// TIA Portal V20 export
FUNCTION "CollectAlarms" : Void   // FC62, LAD
TITLE = Alarm Collector Unit
// Collects alarms from the respective level and categorises the alarms into the different alarm classes.
// stored: Namespace Unit1, SetENOAutomatically false
   VAR_INPUT
      resetAlarms : Bool;
      disableAlarms : Bool;
   END_VAR
   VAR_OUTPUT
      commandsToUnit : "LUC_typeStateCommands";   // Feedback to the unit
   END_VAR
   VAR CONSTANT
      DelayTime : Time := T#300ms;
      TRUE : Bool := TRUE;
      FALSE : Bool;
   END_VAR
BEGIN

REGION Network 1: Reset Alarms
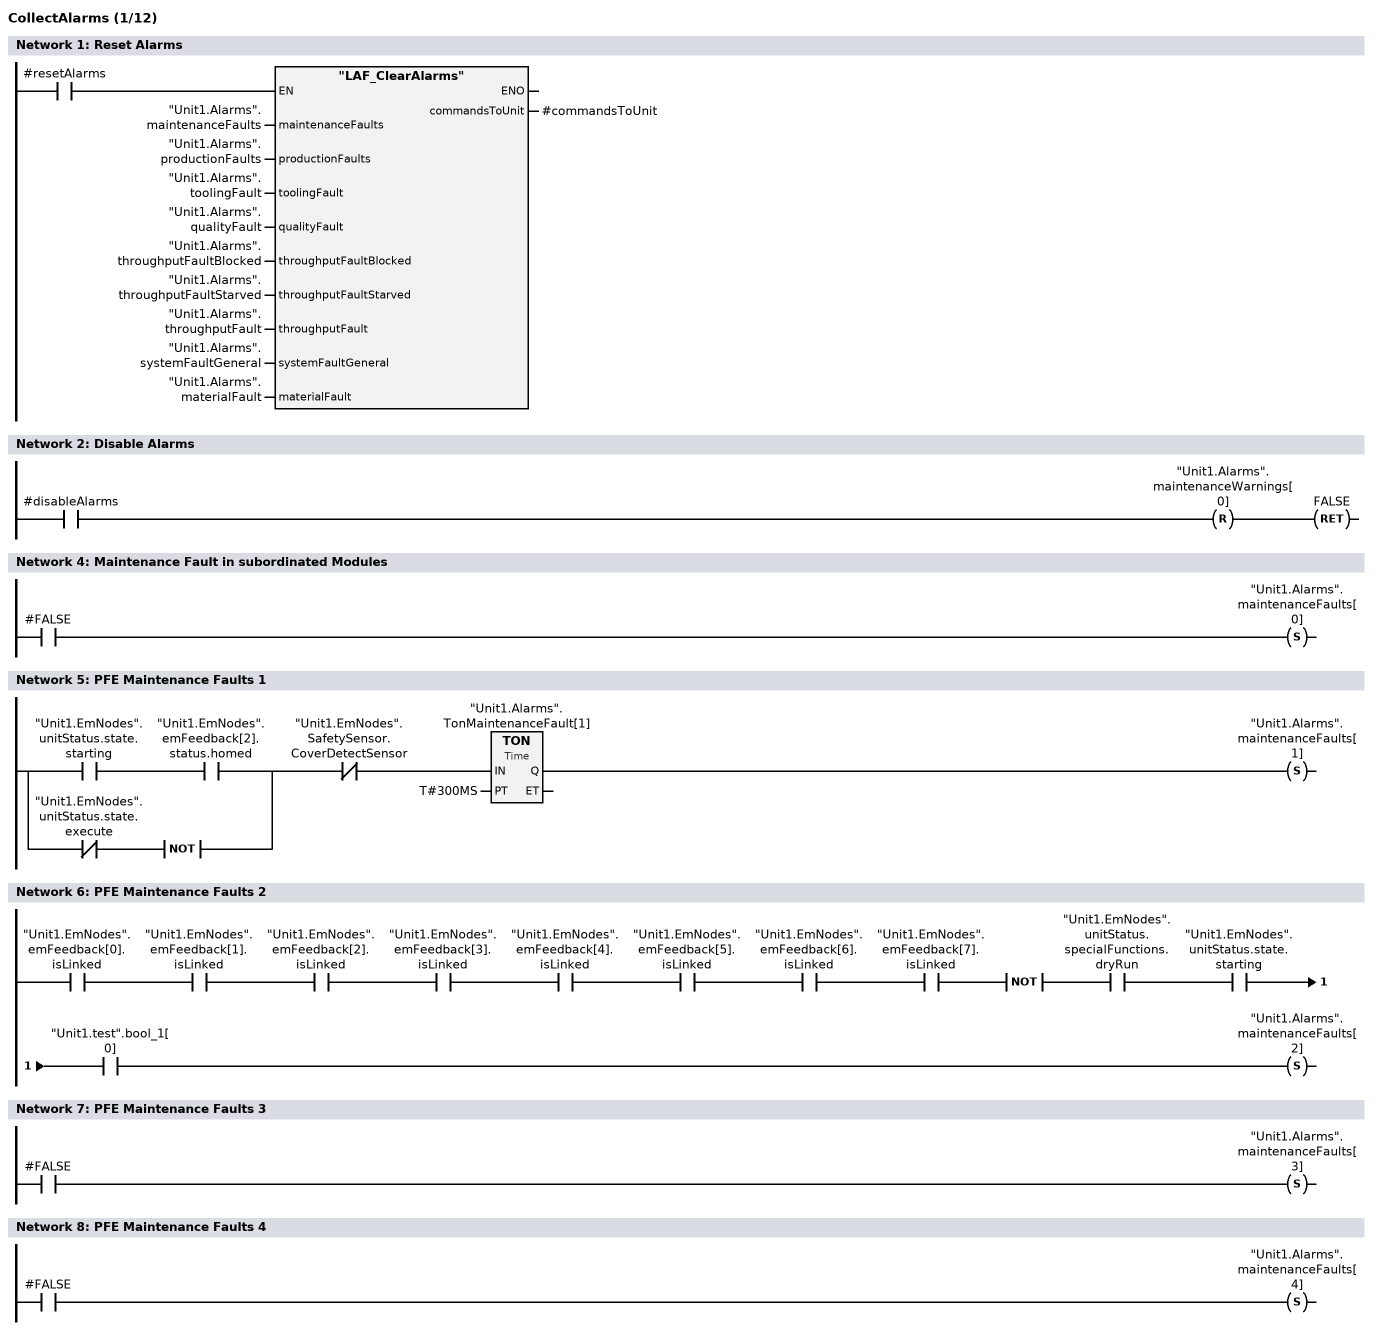
   RUNG wire#powerrail
      Contact( #resetAlarms )
      "LAF_ClearAlarms"(maintenanceFaults := "Unit1.Alarms".maintenanceFaults, productionFaults := "Unit1.Alarms".productionFaults, toolingFault := "Unit1.Alarms".toolingFault, qualityFault := "Unit1.Alarms".qualityFault, throughputFaultBlocked := "Unit1.Alarms".throughputFaultBlocked, throughputFaultStarved := "Unit1.Alarms".throughputFaultStarved, throughputFault := "Unit1.Alarms".throughputFault, systemFaultGeneral := "Unit1.Alarms".systemFaultGeneral, materialFault := "Unit1.Alarms".materialFault, commandsToUnit => #commandsToUnit)
   END_RUNG
   // the same network as SCL:
   IF #resetAlarms THEN
       "LAF_ClearAlarms"(maintenanceFaults := "Unit1.Alarms".maintenanceFaults,
                         productionFaults := "Unit1.Alarms".productionFaults,
                         toolingFault := "Unit1.Alarms".toolingFault,
                         qualityFault := "Unit1.Alarms".qualityFault,
                         throughputFaultBlocked := "Unit1.Alarms".throughputFaultBlocked,
                         throughputFaultStarved := "Unit1.Alarms".throughputFaultStarved,
                         throughputFault := "Unit1.Alarms".throughputFault,
                         systemFaultGeneral := "Unit1.Alarms".systemFaultGeneral,
                         materialFault := "Unit1.Alarms".materialFault,
                         commandsToUnit => #commandsToUnit);
   END_IF;
END_REGION

REGION Network 2: Disable Alarms
   RUNG wire#powerrail
      Contact( #disableAlarms )
      R_Coil( "Unit1.Alarms".maintenanceWarnings[0] )
      ReturnCoil( FALSE )
   END_RUNG
   // the same network as SCL:
   IF #disableAlarms THEN
       "Unit1.Alarms".maintenanceWarnings[0] := FALSE;
       ENO := FALSE;
       RETURN;
   END_IF;
END_REGION

REGION Network 3: *************** Fault ************************
END_REGION

REGION Network 4: Maintenance Fault in subordinated Modules
   RUNG wire#powerrail
      Contact( #FALSE )
      S_Coil( "Unit1.Alarms".maintenanceFaults[0] )
   END_RUNG
   // the same network as SCL:
   IF #FALSE THEN "Unit1.Alarms".maintenanceFaults[0] := TRUE; END_IF;
END_REGION

REGION Network 5: PFE Maintenance Faults 1
   RUNG wire#powerrail
      Contact( "Unit1.EmNodes".unitStatus.state.starting )
      Contact( "Unit1.EmNodes".emFeedback[2].status.homed )
      wire#w1
      I_Contact( "Unit1.EmNodes".SafetySensor.CoverDetectSensor )
      { S7_Templates := "time_type := Time" } "Unit1.Alarms".TonMaintenanceFault[1].TON(pt := T#300MS, et =>)
      S_Coil( "Unit1.Alarms".maintenanceFaults[1] )
   END_RUNG
   RUNG wire#powerrail
      I_Contact( "Unit1.EmNodes".unitStatus.state.execute )
      Not()
   END_RUNG wire#w1
   // the same network as SCL:
   "Unit1.Alarms".TonMaintenanceFault[1].TON(IN := (("Unit1.EmNodes".unitStatus.state.starting AND "Unit1.EmNodes".emFeedback[2].status.homed) OR NOT (NOT "Unit1.EmNodes".unitStatus.state.execute)) AND NOT "Unit1.EmNodes".SafetySensor.CoverDetectSensor,
                           PT := T#300MS);
   IF "Unit1.Alarms".TonMaintenanceFault[1].Q THEN "Unit1.Alarms".maintenanceFaults[1] := TRUE; END_IF;
END_REGION

REGION Network 6: PFE Maintenance Faults 2
   RUNG wire#powerrail
      Contact( "Unit1.EmNodes".emFeedback[0].isLinked )
      Contact( "Unit1.EmNodes".emFeedback[1].isLinked )
      Contact( "Unit1.EmNodes".emFeedback[2].isLinked )
      Contact( "Unit1.EmNodes".emFeedback[3].isLinked )
      Contact( "Unit1.EmNodes".emFeedback[4].isLinked )
      Contact( "Unit1.EmNodes".emFeedback[5].isLinked )
      Contact( "Unit1.EmNodes".emFeedback[6].isLinked )
      Contact( "Unit1.EmNodes".emFeedback[7].isLinked )
      Not()
      Contact( "Unit1.EmNodes".unitStatus.specialFunctions.dryRun )
      Contact( "Unit1.EmNodes".unitStatus.state.starting )
      Contact( "Unit1.test".bool_1[0] )
      S_Coil( "Unit1.Alarms".maintenanceFaults[2] )
   END_RUNG
   // the same network as SCL:
   IF NOT ("Unit1.EmNodes".emFeedback[0].isLinked AND "Unit1.EmNodes".emFeedback[1].isLinked AND "Unit1.EmNodes".emFeedback[2].isLinked AND "Unit1.EmNodes".emFeedback[3].isLinked AND "Unit1.EmNodes".emFeedback[4].isLinked AND "Unit1.EmNodes".emFeedback[5].isLinked AND "Unit1.EmNodes".emFeedback[6].isLinked AND "Unit1.EmNodes".emFeedback[7].isLinked) AND "Unit1.EmNodes".unitStatus.specialFunctions.dryRun AND "Unit1.EmNodes".unitStatus.state.starting AND "Unit1.test".bool_1[0] THEN
       "Unit1.Alarms".maintenanceFaults[2] := TRUE;
   END_IF;
END_REGION

REGION Network 7: PFE Maintenance Faults 3
   RUNG wire#powerrail
      Contact( #FALSE )
      S_Coil( "Unit1.Alarms".maintenanceFaults[3] )
   END_RUNG
   // the same network as SCL:
   IF #FALSE THEN "Unit1.Alarms".maintenanceFaults[3] := TRUE; END_IF;
END_REGION

REGION Network 8: PFE Maintenance Faults 4
   RUNG wire#powerrail
      Contact( #FALSE )
      S_Coil( "Unit1.Alarms".maintenanceFaults[4] )
   END_RUNG
   // the same network as SCL:
   IF #FALSE THEN "Unit1.Alarms".maintenanceFaults[4] := TRUE; END_IF;
END_REGION

REGION Network 9: PFE Maintenance Faults 5
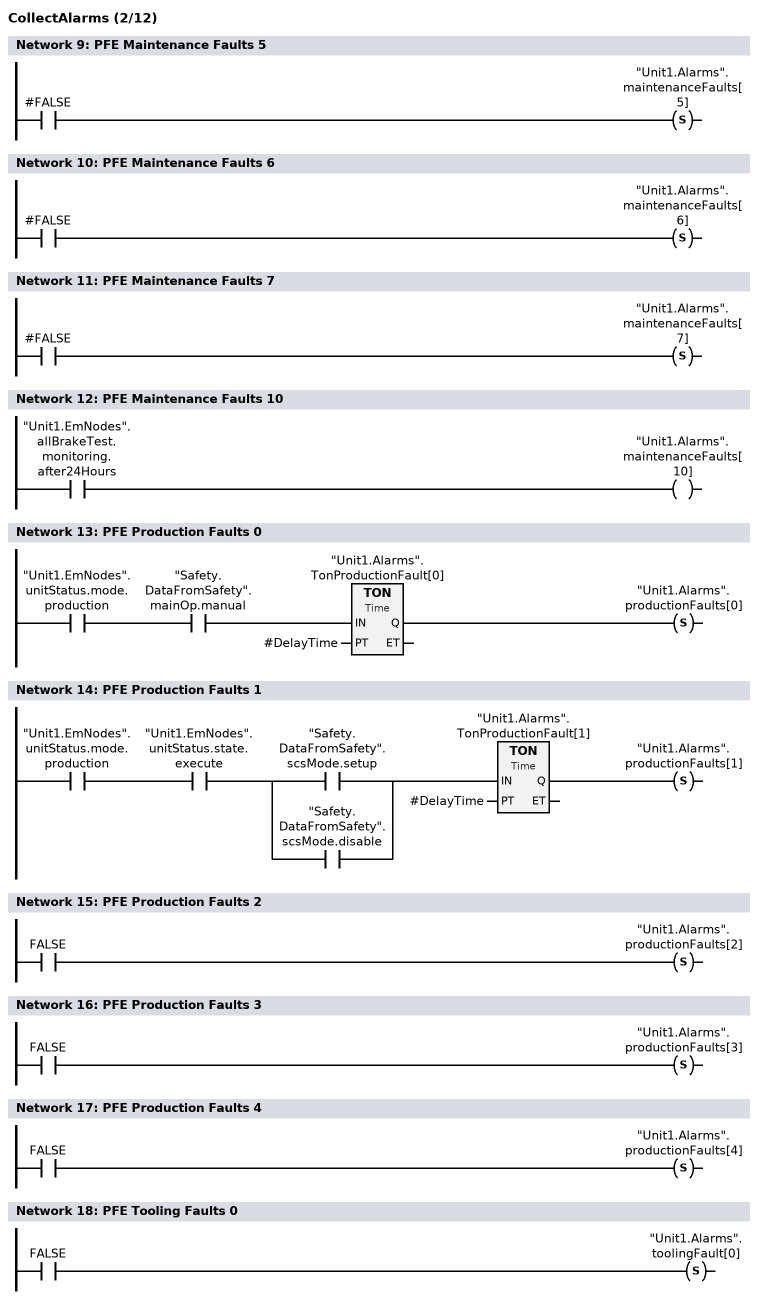
   RUNG wire#powerrail
      Contact( #FALSE )
      S_Coil( "Unit1.Alarms".maintenanceFaults[5] )
   END_RUNG
   // the same network as SCL:
   IF #FALSE THEN "Unit1.Alarms".maintenanceFaults[5] := TRUE; END_IF;
END_REGION

REGION Network 10: PFE Maintenance Faults 6
   RUNG wire#powerrail
      Contact( #FALSE )
      S_Coil( "Unit1.Alarms".maintenanceFaults[6] )
   END_RUNG
   // the same network as SCL:
   IF #FALSE THEN "Unit1.Alarms".maintenanceFaults[6] := TRUE; END_IF;
END_REGION

REGION Network 11: PFE Maintenance Faults 7
   RUNG wire#powerrail
      Contact( #FALSE )
      S_Coil( "Unit1.Alarms".maintenanceFaults[7] )
   END_RUNG
   // the same network as SCL:
   IF #FALSE THEN "Unit1.Alarms".maintenanceFaults[7] := TRUE; END_IF;
END_REGION

REGION Network 12: PFE Maintenance Faults 10
   RUNG wire#powerrail
      Contact( "Unit1.EmNodes".allBrakeTest.monitoring.after24Hours )
      Coil( "Unit1.Alarms".maintenanceFaults[10] )
   END_RUNG
   // the same network as SCL:
   "Unit1.Alarms".maintenanceFaults[10] := "Unit1.EmNodes".allBrakeTest.monitoring.after24Hours;
END_REGION

REGION Network 13: PFE Production Faults 0
   RUNG wire#powerrail
      Contact( "Unit1.EmNodes".unitStatus.mode.production )
      Contact( "Safety.DataFromSafety".mainOp.manual )
      { S7_Templates := "time_type := Time" } "Unit1.Alarms".TonProductionFault[0].TON(pt := #DelayTime, et =>)
      S_Coil( "Unit1.Alarms".productionFaults[0] )
   END_RUNG
   // the same network as SCL:
   "Unit1.Alarms".TonProductionFault[0].TON(IN := "Unit1.EmNodes".unitStatus.mode.production AND "Safety.DataFromSafety".mainOp.manual,
                           PT := #DelayTime);
   IF "Unit1.Alarms".TonProductionFault[0].Q THEN "Unit1.Alarms".productionFaults[0] := TRUE; END_IF;
END_REGION

REGION Network 14: PFE Production Faults 1
   RUNG wire#powerrail
      Contact( "Unit1.EmNodes".unitStatus.mode.production )
      Contact( "Unit1.EmNodes".unitStatus.state.execute )
      wire#w1
      Contact( "Safety.DataFromSafety".scsMode.setup )
      wire#w2
      { S7_Templates := "time_type := Time" } "Unit1.Alarms".TonProductionFault[1].TON(pt := #DelayTime, et =>)
      S_Coil( "Unit1.Alarms".productionFaults[1] )
   END_RUNG
   RUNG wire#w1
      Contact( "Safety.DataFromSafety".scsMode.disable )
   END_RUNG wire#w2
   // the same network as SCL:
   "Unit1.Alarms".TonProductionFault[1].TON(IN := "Unit1.EmNodes".unitStatus.mode.production AND "Unit1.EmNodes".unitStatus.state.execute AND ("Safety.DataFromSafety".scsMode.setup OR "Safety.DataFromSafety".scsMode.disable),
                           PT := #DelayTime);
   IF "Unit1.Alarms".TonProductionFault[1].Q THEN "Unit1.Alarms".productionFaults[1] := TRUE; END_IF;
END_REGION

REGION Network 15: PFE Production Faults 2
   RUNG wire#powerrail
      Contact( FALSE )
      S_Coil( "Unit1.Alarms".productionFaults[2] )
   END_RUNG
   // the same network as SCL:
   IF FALSE THEN "Unit1.Alarms".productionFaults[2] := TRUE; END_IF;
END_REGION

REGION Network 16: PFE Production Faults 3
   RUNG wire#powerrail
      Contact( FALSE )
      S_Coil( "Unit1.Alarms".productionFaults[3] )
   END_RUNG
   // the same network as SCL:
   IF FALSE THEN "Unit1.Alarms".productionFaults[3] := TRUE; END_IF;
END_REGION

REGION Network 17: PFE Production Faults 4
   RUNG wire#powerrail
      Contact( FALSE )
      S_Coil( "Unit1.Alarms".productionFaults[4] )
   END_RUNG
   // the same network as SCL:
   IF FALSE THEN "Unit1.Alarms".productionFaults[4] := TRUE; END_IF;
END_REGION

REGION Network 18: PFE Tooling Faults 0
   RUNG wire#powerrail
      Contact( FALSE )
      S_Coil( "Unit1.Alarms".toolingFault[0] )
   END_RUNG
   // the same network as SCL:
   IF FALSE THEN "Unit1.Alarms".toolingFault[0] := TRUE; END_IF;
END_REGION

REGION Network 19: PFE Tooling Faults 1
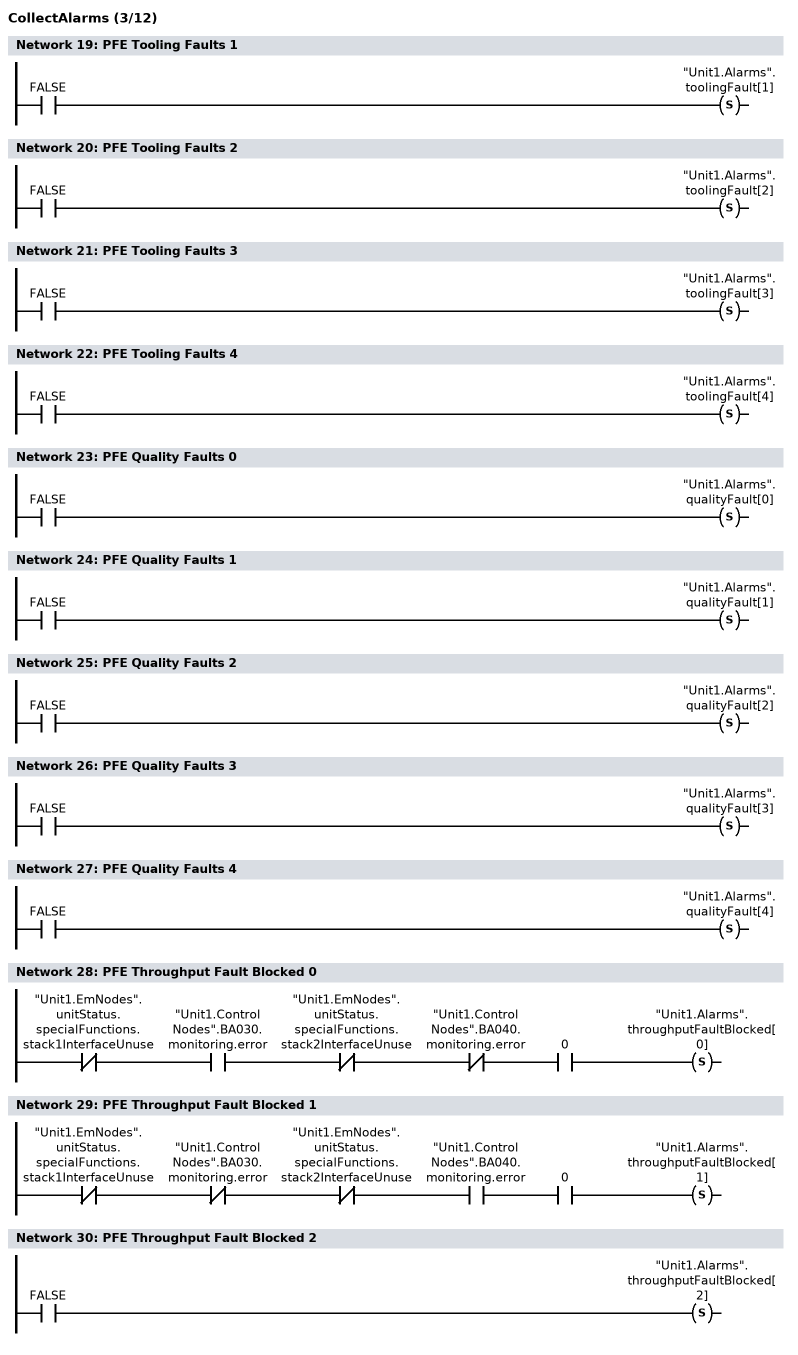
   RUNG wire#powerrail
      Contact( FALSE )
      S_Coil( "Unit1.Alarms".toolingFault[1] )
   END_RUNG
   // the same network as SCL:
   IF FALSE THEN "Unit1.Alarms".toolingFault[1] := TRUE; END_IF;
END_REGION

REGION Network 20: PFE Tooling Faults 2
   RUNG wire#powerrail
      Contact( FALSE )
      S_Coil( "Unit1.Alarms".toolingFault[2] )
   END_RUNG
   // the same network as SCL:
   IF FALSE THEN "Unit1.Alarms".toolingFault[2] := TRUE; END_IF;
END_REGION

REGION Network 21: PFE Tooling Faults 3
   RUNG wire#powerrail
      Contact( FALSE )
      S_Coil( "Unit1.Alarms".toolingFault[3] )
   END_RUNG
   // the same network as SCL:
   IF FALSE THEN "Unit1.Alarms".toolingFault[3] := TRUE; END_IF;
END_REGION

REGION Network 22: PFE Tooling Faults 4
   RUNG wire#powerrail
      Contact( FALSE )
      S_Coil( "Unit1.Alarms".toolingFault[4] )
   END_RUNG
   // the same network as SCL:
   IF FALSE THEN "Unit1.Alarms".toolingFault[4] := TRUE; END_IF;
END_REGION

REGION Network 23: PFE Quality Faults 0
   RUNG wire#powerrail
      Contact( FALSE )
      S_Coil( "Unit1.Alarms".qualityFault[0] )
   END_RUNG
   // the same network as SCL:
   IF FALSE THEN "Unit1.Alarms".qualityFault[0] := TRUE; END_IF;
END_REGION

REGION Network 24: PFE Quality Faults 1
   RUNG wire#powerrail
      Contact( FALSE )
      S_Coil( "Unit1.Alarms".qualityFault[1] )
   END_RUNG
   // the same network as SCL:
   IF FALSE THEN "Unit1.Alarms".qualityFault[1] := TRUE; END_IF;
END_REGION

REGION Network 25: PFE Quality Faults 2
   RUNG wire#powerrail
      Contact( FALSE )
      S_Coil( "Unit1.Alarms".qualityFault[2] )
   END_RUNG
   // the same network as SCL:
   IF FALSE THEN "Unit1.Alarms".qualityFault[2] := TRUE; END_IF;
END_REGION

REGION Network 26: PFE Quality Faults 3
   RUNG wire#powerrail
      Contact( FALSE )
      S_Coil( "Unit1.Alarms".qualityFault[3] )
   END_RUNG
   // the same network as SCL:
   IF FALSE THEN "Unit1.Alarms".qualityFault[3] := TRUE; END_IF;
END_REGION

REGION Network 27: PFE Quality Faults 4
   RUNG wire#powerrail
      Contact( FALSE )
      S_Coil( "Unit1.Alarms".qualityFault[4] )
   END_RUNG
   // the same network as SCL:
   IF FALSE THEN "Unit1.Alarms".qualityFault[4] := TRUE; END_IF;
END_REGION

REGION Network 28: PFE Throughput Fault Blocked 0
   RUNG wire#powerrail
      I_Contact( "Unit1.EmNodes".unitStatus.specialFunctions.stack1InterfaceUnuse )
      Contact( "Unit1.ControlNodes".BA030.monitoring.error )
      I_Contact( "Unit1.EmNodes".unitStatus.specialFunctions.stack2InterfaceUnuse )
      I_Contact( "Unit1.ControlNodes".BA040.monitoring.error )
      Contact( 0 )
      S_Coil( "Unit1.Alarms".throughputFaultBlocked[0] )
   END_RUNG
   // the same network as SCL:
   IF NOT "Unit1.EmNodes".unitStatus.specialFunctions.stack1InterfaceUnuse AND "Unit1.ControlNodes".BA030.monitoring.error AND NOT "Unit1.EmNodes".unitStatus.specialFunctions.stack2InterfaceUnuse AND NOT "Unit1.ControlNodes".BA040.monitoring.error AND 0 THEN
       "Unit1.Alarms".throughputFaultBlocked[0] := TRUE;
   END_IF;
END_REGION

REGION Network 29: PFE Throughput Fault Blocked 1
   RUNG wire#powerrail
      I_Contact( "Unit1.EmNodes".unitStatus.specialFunctions.stack1InterfaceUnuse )
      I_Contact( "Unit1.ControlNodes".BA030.monitoring.error )
      I_Contact( "Unit1.EmNodes".unitStatus.specialFunctions.stack2InterfaceUnuse )
      Contact( "Unit1.ControlNodes".BA040.monitoring.error )
      Contact( 0 )
      S_Coil( "Unit1.Alarms".throughputFaultBlocked[1] )
   END_RUNG
   // the same network as SCL:
   IF NOT "Unit1.EmNodes".unitStatus.specialFunctions.stack1InterfaceUnuse AND NOT "Unit1.ControlNodes".BA030.monitoring.error AND NOT "Unit1.EmNodes".unitStatus.specialFunctions.stack2InterfaceUnuse AND "Unit1.ControlNodes".BA040.monitoring.error AND 0 THEN
       "Unit1.Alarms".throughputFaultBlocked[1] := TRUE;
   END_IF;
END_REGION

REGION Network 30: PFE Throughput Fault Blocked 2
   RUNG wire#powerrail
      Contact( FALSE )
      S_Coil( "Unit1.Alarms".throughputFaultBlocked[2] )
   END_RUNG
   // the same network as SCL:
   IF FALSE THEN "Unit1.Alarms".throughputFaultBlocked[2] := TRUE; END_IF;
END_REGION

REGION Network 31: PFE Throughput Fault Blocked 3
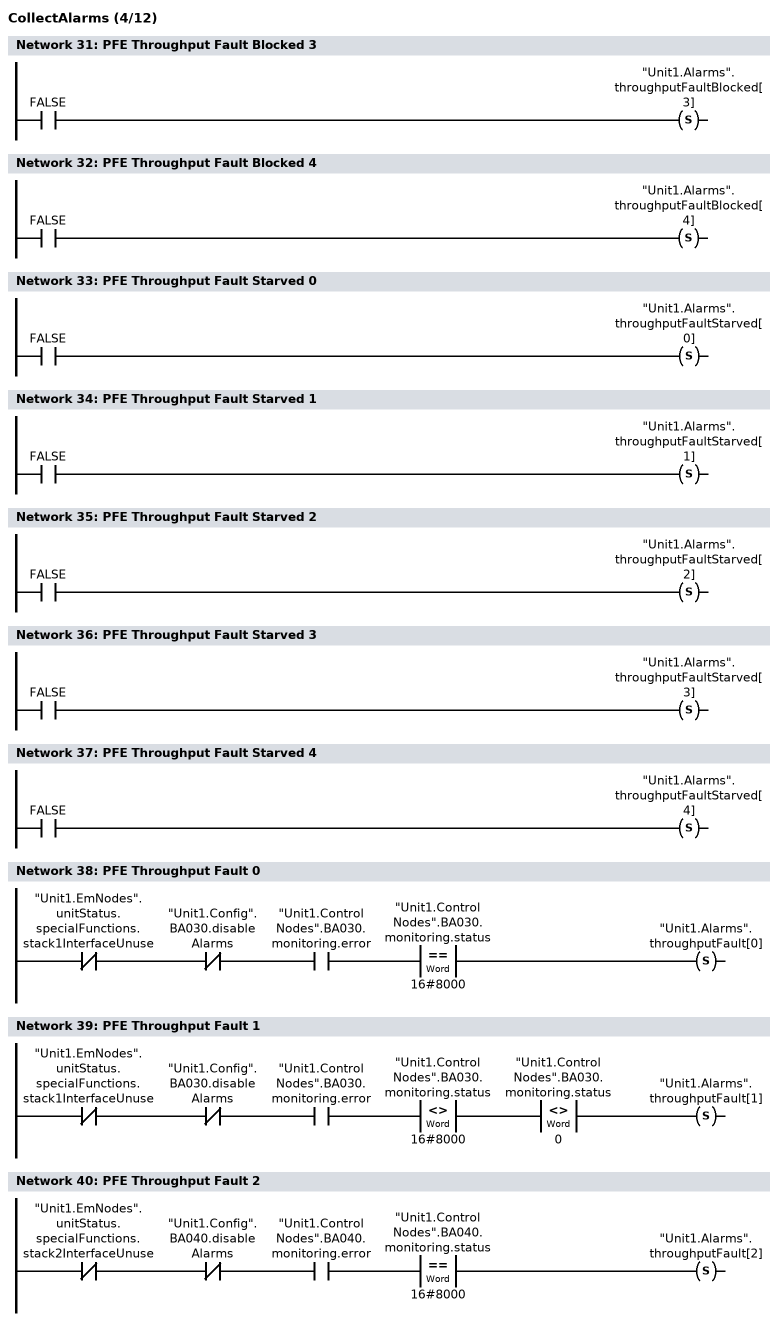
   RUNG wire#powerrail
      Contact( FALSE )
      S_Coil( "Unit1.Alarms".throughputFaultBlocked[3] )
   END_RUNG
   // the same network as SCL:
   IF FALSE THEN "Unit1.Alarms".throughputFaultBlocked[3] := TRUE; END_IF;
END_REGION

REGION Network 32: PFE Throughput Fault Blocked 4
   RUNG wire#powerrail
      Contact( FALSE )
      S_Coil( "Unit1.Alarms".throughputFaultBlocked[4] )
   END_RUNG
   // the same network as SCL:
   IF FALSE THEN "Unit1.Alarms".throughputFaultBlocked[4] := TRUE; END_IF;
END_REGION

REGION Network 33: PFE Throughput Fault Starved 0
   RUNG wire#powerrail
      Contact( FALSE )
      S_Coil( "Unit1.Alarms".throughputFaultStarved[0] )
   END_RUNG
   // the same network as SCL:
   IF FALSE THEN "Unit1.Alarms".throughputFaultStarved[0] := TRUE; END_IF;
END_REGION

REGION Network 34: PFE Throughput Fault Starved 1
   RUNG wire#powerrail
      Contact( FALSE )
      S_Coil( "Unit1.Alarms".throughputFaultStarved[1] )
   END_RUNG
   // the same network as SCL:
   IF FALSE THEN "Unit1.Alarms".throughputFaultStarved[1] := TRUE; END_IF;
END_REGION

REGION Network 35: PFE Throughput Fault Starved 2
   RUNG wire#powerrail
      Contact( FALSE )
      S_Coil( "Unit1.Alarms".throughputFaultStarved[2] )
   END_RUNG
   // the same network as SCL:
   IF FALSE THEN "Unit1.Alarms".throughputFaultStarved[2] := TRUE; END_IF;
END_REGION

REGION Network 36: PFE Throughput Fault Starved 3
   RUNG wire#powerrail
      Contact( FALSE )
      S_Coil( "Unit1.Alarms".throughputFaultStarved[3] )
   END_RUNG
   // the same network as SCL:
   IF FALSE THEN "Unit1.Alarms".throughputFaultStarved[3] := TRUE; END_IF;
END_REGION

REGION Network 37: PFE Throughput Fault Starved 4
   RUNG wire#powerrail
      Contact( FALSE )
      S_Coil( "Unit1.Alarms".throughputFaultStarved[4] )
   END_RUNG
   // the same network as SCL:
   IF FALSE THEN "Unit1.Alarms".throughputFaultStarved[4] := TRUE; END_IF;
END_REGION

REGION Network 38: PFE Throughput Fault 0
   RUNG wire#powerrail
      I_Contact( "Unit1.EmNodes".unitStatus.specialFunctions.stack1InterfaceUnuse )
      I_Contact( "Unit1.Config".BA030.disableAlarms )
      Contact( "Unit1.ControlNodes".BA030.monitoring.error )
      { S7_Templates := "SrcType := Word" } EQ_Contact(in1 := "Unit1.ControlNodes".BA030.monitoring.status, in2 := 16#8000)
      S_Coil( "Unit1.Alarms".throughputFault[0] )
   END_RUNG
   // the same network as SCL:
   IF NOT "Unit1.EmNodes".unitStatus.specialFunctions.stack1InterfaceUnuse AND NOT "Unit1.Config".BA030.disableAlarms AND "Unit1.ControlNodes".BA030.monitoring.error AND ("Unit1.ControlNodes".BA030.monitoring.status = 16#8000) THEN
       "Unit1.Alarms".throughputFault[0] := TRUE;
   END_IF;
END_REGION

REGION Network 39: PFE Throughput Fault 1
   RUNG wire#powerrail
      I_Contact( "Unit1.EmNodes".unitStatus.specialFunctions.stack1InterfaceUnuse )
      I_Contact( "Unit1.Config".BA030.disableAlarms )
      Contact( "Unit1.ControlNodes".BA030.monitoring.error )
      { S7_Templates := "SrcType := Word" } NE_Contact(in1 := "Unit1.ControlNodes".BA030.monitoring.status, in2 := 16#8000)
      { S7_Templates := "SrcType := Word" } NE_Contact(in1 := "Unit1.ControlNodes".BA030.monitoring.status, in2 := 0)
      S_Coil( "Unit1.Alarms".throughputFault[1] )
   END_RUNG
   // the same network as SCL:
   IF NOT "Unit1.EmNodes".unitStatus.specialFunctions.stack1InterfaceUnuse AND NOT "Unit1.Config".BA030.disableAlarms AND "Unit1.ControlNodes".BA030.monitoring.error AND ("Unit1.ControlNodes".BA030.monitoring.status <> 16#8000) AND ("Unit1.ControlNodes".BA030.monitoring.status <> 0) THEN
       "Unit1.Alarms".throughputFault[1] := TRUE;
   END_IF;
END_REGION

REGION Network 40: PFE Throughput Fault 2
   RUNG wire#powerrail
      I_Contact( "Unit1.EmNodes".unitStatus.specialFunctions.stack2InterfaceUnuse )
      I_Contact( "Unit1.Config".BA040.disableAlarms )
      Contact( "Unit1.ControlNodes".BA040.monitoring.error )
      { S7_Templates := "SrcType := Word" } EQ_Contact(in1 := "Unit1.ControlNodes".BA040.monitoring.status, in2 := 16#8000)
      S_Coil( "Unit1.Alarms".throughputFault[2] )
   END_RUNG
   // the same network as SCL:
   IF NOT "Unit1.EmNodes".unitStatus.specialFunctions.stack2InterfaceUnuse AND NOT "Unit1.Config".BA040.disableAlarms AND "Unit1.ControlNodes".BA040.monitoring.error AND ("Unit1.ControlNodes".BA040.monitoring.status = 16#8000) THEN
       "Unit1.Alarms".throughputFault[2] := TRUE;
   END_IF;
END_REGION

REGION Network 41: PFE Throughput Fault 3
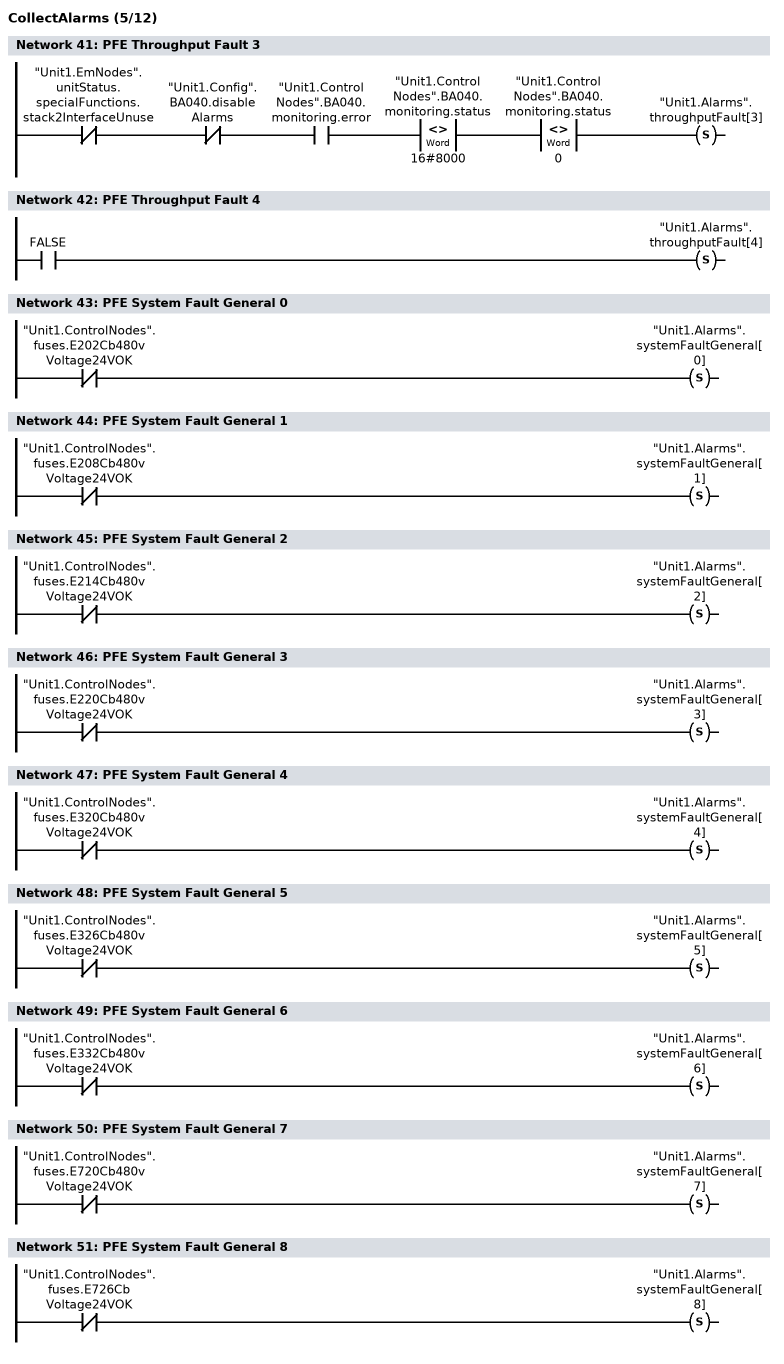
   RUNG wire#powerrail
      I_Contact( "Unit1.EmNodes".unitStatus.specialFunctions.stack2InterfaceUnuse )
      I_Contact( "Unit1.Config".BA040.disableAlarms )
      Contact( "Unit1.ControlNodes".BA040.monitoring.error )
      { S7_Templates := "SrcType := Word" } NE_Contact(in1 := "Unit1.ControlNodes".BA040.monitoring.status, in2 := 16#8000)
      { S7_Templates := "SrcType := Word" } NE_Contact(in1 := "Unit1.ControlNodes".BA040.monitoring.status, in2 := 0)
      S_Coil( "Unit1.Alarms".throughputFault[3] )
   END_RUNG
   // the same network as SCL:
   IF NOT "Unit1.EmNodes".unitStatus.specialFunctions.stack2InterfaceUnuse AND NOT "Unit1.Config".BA040.disableAlarms AND "Unit1.ControlNodes".BA040.monitoring.error AND ("Unit1.ControlNodes".BA040.monitoring.status <> 16#8000) AND ("Unit1.ControlNodes".BA040.monitoring.status <> 0) THEN
       "Unit1.Alarms".throughputFault[3] := TRUE;
   END_IF;
END_REGION

REGION Network 42: PFE Throughput Fault 4
   RUNG wire#powerrail
      Contact( FALSE )
      S_Coil( "Unit1.Alarms".throughputFault[4] )
   END_RUNG
   // the same network as SCL:
   IF FALSE THEN "Unit1.Alarms".throughputFault[4] := TRUE; END_IF;
END_REGION

REGION Network 43: PFE System Fault General 0
   RUNG wire#powerrail
      I_Contact( "Unit1.ControlNodes".fuses.E202Cb480vVoltage24VOK )
      S_Coil( "Unit1.Alarms".systemFaultGeneral[0] )
   END_RUNG
   // the same network as SCL:
   IF NOT "Unit1.ControlNodes".fuses.E202Cb480vVoltage24VOK THEN
       "Unit1.Alarms".systemFaultGeneral[0] := TRUE;
   END_IF;
END_REGION

REGION Network 44: PFE System Fault General 1
   RUNG wire#powerrail
      I_Contact( "Unit1.ControlNodes".fuses.E208Cb480vVoltage24VOK )
      S_Coil( "Unit1.Alarms".systemFaultGeneral[1] )
   END_RUNG
   // the same network as SCL:
   IF NOT "Unit1.ControlNodes".fuses.E208Cb480vVoltage24VOK THEN
       "Unit1.Alarms".systemFaultGeneral[1] := TRUE;
   END_IF;
END_REGION

REGION Network 45: PFE System Fault General 2
   RUNG wire#powerrail
      I_Contact( "Unit1.ControlNodes".fuses.E214Cb480vVoltage24VOK )
      S_Coil( "Unit1.Alarms".systemFaultGeneral[2] )
   END_RUNG
   // the same network as SCL:
   IF NOT "Unit1.ControlNodes".fuses.E214Cb480vVoltage24VOK THEN
       "Unit1.Alarms".systemFaultGeneral[2] := TRUE;
   END_IF;
END_REGION

REGION Network 46: PFE System Fault General 3
   RUNG wire#powerrail
      I_Contact( "Unit1.ControlNodes".fuses.E220Cb480vVoltage24VOK )
      S_Coil( "Unit1.Alarms".systemFaultGeneral[3] )
   END_RUNG
   // the same network as SCL:
   IF NOT "Unit1.ControlNodes".fuses.E220Cb480vVoltage24VOK THEN
       "Unit1.Alarms".systemFaultGeneral[3] := TRUE;
   END_IF;
END_REGION

REGION Network 47: PFE System Fault General 4
   RUNG wire#powerrail
      I_Contact( "Unit1.ControlNodes".fuses.E320Cb480vVoltage24VOK )
      S_Coil( "Unit1.Alarms".systemFaultGeneral[4] )
   END_RUNG
   // the same network as SCL:
   IF NOT "Unit1.ControlNodes".fuses.E320Cb480vVoltage24VOK THEN
       "Unit1.Alarms".systemFaultGeneral[4] := TRUE;
   END_IF;
END_REGION

REGION Network 48: PFE System Fault General 5
   RUNG wire#powerrail
      I_Contact( "Unit1.ControlNodes".fuses.E326Cb480vVoltage24VOK )
      S_Coil( "Unit1.Alarms".systemFaultGeneral[5] )
   END_RUNG
   // the same network as SCL:
   IF NOT "Unit1.ControlNodes".fuses.E326Cb480vVoltage24VOK THEN
       "Unit1.Alarms".systemFaultGeneral[5] := TRUE;
   END_IF;
END_REGION

REGION Network 49: PFE System Fault General 6
   RUNG wire#powerrail
      I_Contact( "Unit1.ControlNodes".fuses.E332Cb480vVoltage24VOK )
      S_Coil( "Unit1.Alarms".systemFaultGeneral[6] )
   END_RUNG
   // the same network as SCL:
   IF NOT "Unit1.ControlNodes".fuses.E332Cb480vVoltage24VOK THEN
       "Unit1.Alarms".systemFaultGeneral[6] := TRUE;
   END_IF;
END_REGION

REGION Network 50: PFE System Fault General 7
   RUNG wire#powerrail
      I_Contact( "Unit1.ControlNodes".fuses.E720Cb480vVoltage24VOK )
      S_Coil( "Unit1.Alarms".systemFaultGeneral[7] )
   END_RUNG
   // the same network as SCL:
   IF NOT "Unit1.ControlNodes".fuses.E720Cb480vVoltage24VOK THEN
       "Unit1.Alarms".systemFaultGeneral[7] := TRUE;
   END_IF;
END_REGION

REGION Network 51: PFE System Fault General 8
   RUNG wire#powerrail
      I_Contact( "Unit1.ControlNodes".fuses.E726CbVoltage24VOK )
      S_Coil( "Unit1.Alarms".systemFaultGeneral[8] )
   END_RUNG
   // the same network as SCL:
   IF NOT "Unit1.ControlNodes".fuses.E726CbVoltage24VOK THEN
       "Unit1.Alarms".systemFaultGeneral[8] := TRUE;
   END_IF;
END_REGION

REGION Network 52: PFE System Fault General 9
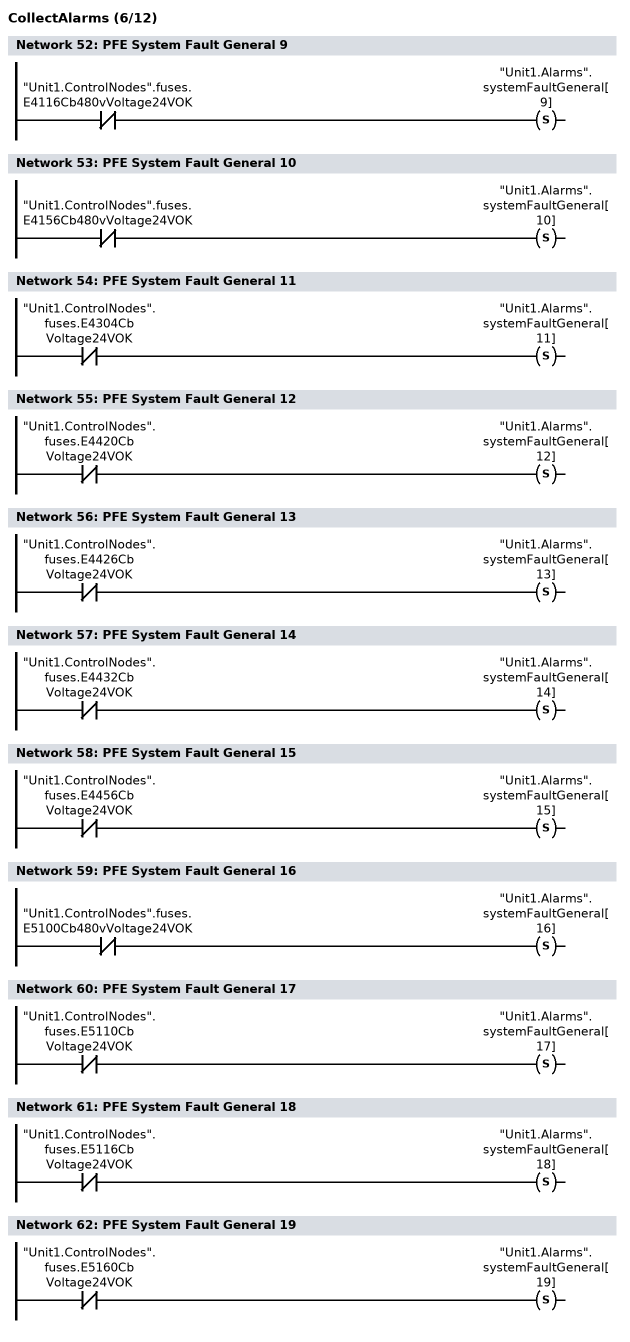
   RUNG wire#powerrail
      I_Contact( "Unit1.ControlNodes".fuses.E4116Cb480vVoltage24VOK )
      S_Coil( "Unit1.Alarms".systemFaultGeneral[9] )
   END_RUNG
   // the same network as SCL:
   IF NOT "Unit1.ControlNodes".fuses.E4116Cb480vVoltage24VOK THEN
       "Unit1.Alarms".systemFaultGeneral[9] := TRUE;
   END_IF;
END_REGION

REGION Network 53: PFE System Fault General 10
   RUNG wire#powerrail
      I_Contact( "Unit1.ControlNodes".fuses.E4156Cb480vVoltage24VOK )
      S_Coil( "Unit1.Alarms".systemFaultGeneral[10] )
   END_RUNG
   // the same network as SCL:
   IF NOT "Unit1.ControlNodes".fuses.E4156Cb480vVoltage24VOK THEN
       "Unit1.Alarms".systemFaultGeneral[10] := TRUE;
   END_IF;
END_REGION

REGION Network 54: PFE System Fault General 11
   RUNG wire#powerrail
      I_Contact( "Unit1.ControlNodes".fuses.E4304CbVoltage24VOK )
      S_Coil( "Unit1.Alarms".systemFaultGeneral[11] )
   END_RUNG
   // the same network as SCL:
   IF NOT "Unit1.ControlNodes".fuses.E4304CbVoltage24VOK THEN
       "Unit1.Alarms".systemFaultGeneral[11] := TRUE;
   END_IF;
END_REGION

REGION Network 55: PFE System Fault General 12
   RUNG wire#powerrail
      I_Contact( "Unit1.ControlNodes".fuses.E4420CbVoltage24VOK )
      S_Coil( "Unit1.Alarms".systemFaultGeneral[12] )
   END_RUNG
   // the same network as SCL:
   IF NOT "Unit1.ControlNodes".fuses.E4420CbVoltage24VOK THEN
       "Unit1.Alarms".systemFaultGeneral[12] := TRUE;
   END_IF;
END_REGION

REGION Network 56: PFE System Fault General 13
   RUNG wire#powerrail
      I_Contact( "Unit1.ControlNodes".fuses.E4426CbVoltage24VOK )
      S_Coil( "Unit1.Alarms".systemFaultGeneral[13] )
   END_RUNG
   // the same network as SCL:
   IF NOT "Unit1.ControlNodes".fuses.E4426CbVoltage24VOK THEN
       "Unit1.Alarms".systemFaultGeneral[13] := TRUE;
   END_IF;
END_REGION

REGION Network 57: PFE System Fault General 14
   RUNG wire#powerrail
      I_Contact( "Unit1.ControlNodes".fuses.E4432CbVoltage24VOK )
      S_Coil( "Unit1.Alarms".systemFaultGeneral[14] )
   END_RUNG
   // the same network as SCL:
   IF NOT "Unit1.ControlNodes".fuses.E4432CbVoltage24VOK THEN
       "Unit1.Alarms".systemFaultGeneral[14] := TRUE;
   END_IF;
END_REGION

REGION Network 58: PFE System Fault General 15
   RUNG wire#powerrail
      I_Contact( "Unit1.ControlNodes".fuses.E4456CbVoltage24VOK )
      S_Coil( "Unit1.Alarms".systemFaultGeneral[15] )
   END_RUNG
   // the same network as SCL:
   IF NOT "Unit1.ControlNodes".fuses.E4456CbVoltage24VOK THEN
       "Unit1.Alarms".systemFaultGeneral[15] := TRUE;
   END_IF;
END_REGION

REGION Network 59: PFE System Fault General 16
   RUNG wire#powerrail
      I_Contact( "Unit1.ControlNodes".fuses.E5100Cb480vVoltage24VOK )
      S_Coil( "Unit1.Alarms".systemFaultGeneral[16] )
   END_RUNG
   // the same network as SCL:
   IF NOT "Unit1.ControlNodes".fuses.E5100Cb480vVoltage24VOK THEN
       "Unit1.Alarms".systemFaultGeneral[16] := TRUE;
   END_IF;
END_REGION

REGION Network 60: PFE System Fault General 17
   RUNG wire#powerrail
      I_Contact( "Unit1.ControlNodes".fuses.E5110CbVoltage24VOK )
      S_Coil( "Unit1.Alarms".systemFaultGeneral[17] )
   END_RUNG
   // the same network as SCL:
   IF NOT "Unit1.ControlNodes".fuses.E5110CbVoltage24VOK THEN
       "Unit1.Alarms".systemFaultGeneral[17] := TRUE;
   END_IF;
END_REGION

REGION Network 61: PFE System Fault General 18
   RUNG wire#powerrail
      I_Contact( "Unit1.ControlNodes".fuses.E5116CbVoltage24VOK )
      S_Coil( "Unit1.Alarms".systemFaultGeneral[18] )
   END_RUNG
   // the same network as SCL:
   IF NOT "Unit1.ControlNodes".fuses.E5116CbVoltage24VOK THEN
       "Unit1.Alarms".systemFaultGeneral[18] := TRUE;
   END_IF;
END_REGION

REGION Network 62: PFE System Fault General 19
   RUNG wire#powerrail
      I_Contact( "Unit1.ControlNodes".fuses.E5160CbVoltage24VOK )
      S_Coil( "Unit1.Alarms".systemFaultGeneral[19] )
   END_RUNG
   // the same network as SCL:
   IF NOT "Unit1.ControlNodes".fuses.E5160CbVoltage24VOK THEN
       "Unit1.Alarms".systemFaultGeneral[19] := TRUE;
   END_IF;
END_REGION

REGION Network 63: PFE System Fault General 20
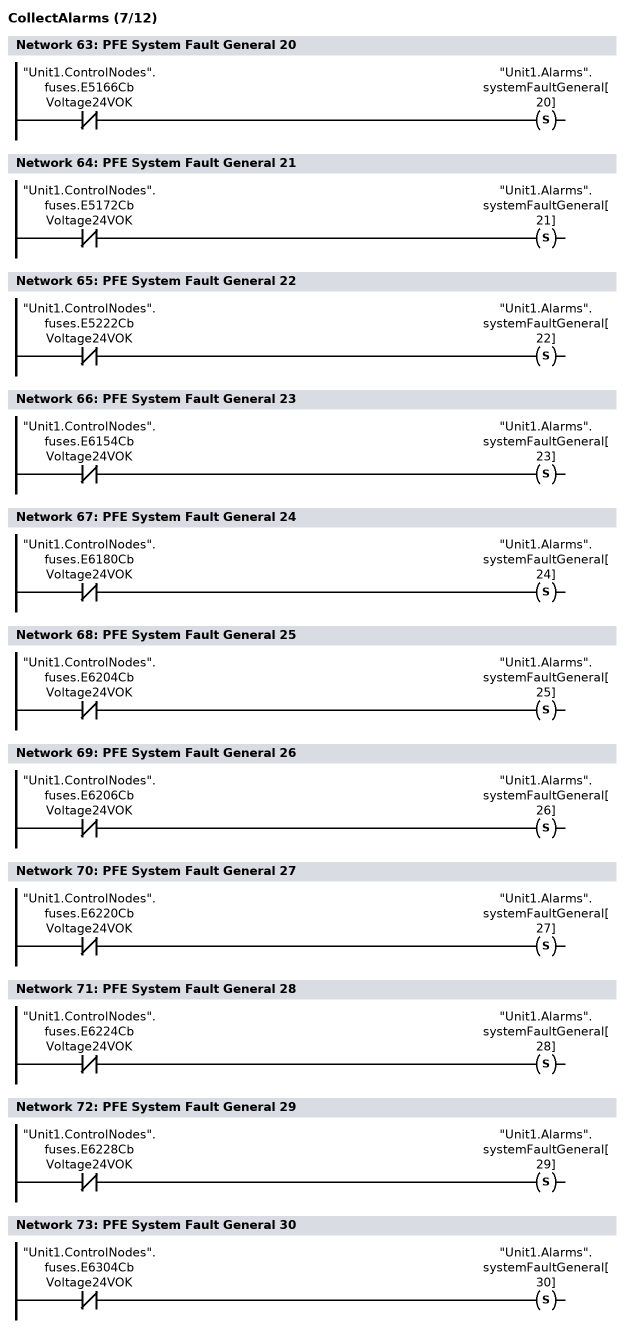
   RUNG wire#powerrail
      I_Contact( "Unit1.ControlNodes".fuses.E5166CbVoltage24VOK )
      S_Coil( "Unit1.Alarms".systemFaultGeneral[20] )
   END_RUNG
   // the same network as SCL:
   IF NOT "Unit1.ControlNodes".fuses.E5166CbVoltage24VOK THEN
       "Unit1.Alarms".systemFaultGeneral[20] := TRUE;
   END_IF;
END_REGION

REGION Network 64: PFE System Fault General 21
   RUNG wire#powerrail
      I_Contact( "Unit1.ControlNodes".fuses.E5172CbVoltage24VOK )
      S_Coil( "Unit1.Alarms".systemFaultGeneral[21] )
   END_RUNG
   // the same network as SCL:
   IF NOT "Unit1.ControlNodes".fuses.E5172CbVoltage24VOK THEN
       "Unit1.Alarms".systemFaultGeneral[21] := TRUE;
   END_IF;
END_REGION

REGION Network 65: PFE System Fault General 22
   RUNG wire#powerrail
      I_Contact( "Unit1.ControlNodes".fuses.E5222CbVoltage24VOK )
      S_Coil( "Unit1.Alarms".systemFaultGeneral[22] )
   END_RUNG
   // the same network as SCL:
   IF NOT "Unit1.ControlNodes".fuses.E5222CbVoltage24VOK THEN
       "Unit1.Alarms".systemFaultGeneral[22] := TRUE;
   END_IF;
END_REGION

REGION Network 66: PFE System Fault General 23
   RUNG wire#powerrail
      I_Contact( "Unit1.ControlNodes".fuses.E6154CbVoltage24VOK )
      S_Coil( "Unit1.Alarms".systemFaultGeneral[23] )
   END_RUNG
   // the same network as SCL:
   IF NOT "Unit1.ControlNodes".fuses.E6154CbVoltage24VOK THEN
       "Unit1.Alarms".systemFaultGeneral[23] := TRUE;
   END_IF;
END_REGION

REGION Network 67: PFE System Fault General 24
   RUNG wire#powerrail
      I_Contact( "Unit1.ControlNodes".fuses.E6180CbVoltage24VOK )
      S_Coil( "Unit1.Alarms".systemFaultGeneral[24] )
   END_RUNG
   // the same network as SCL:
   IF NOT "Unit1.ControlNodes".fuses.E6180CbVoltage24VOK THEN
       "Unit1.Alarms".systemFaultGeneral[24] := TRUE;
   END_IF;
END_REGION

REGION Network 68: PFE System Fault General 25
   RUNG wire#powerrail
      I_Contact( "Unit1.ControlNodes".fuses.E6204CbVoltage24VOK )
      S_Coil( "Unit1.Alarms".systemFaultGeneral[25] )
   END_RUNG
   // the same network as SCL:
   IF NOT "Unit1.ControlNodes".fuses.E6204CbVoltage24VOK THEN
       "Unit1.Alarms".systemFaultGeneral[25] := TRUE;
   END_IF;
END_REGION

REGION Network 69: PFE System Fault General 26
   RUNG wire#powerrail
      I_Contact( "Unit1.ControlNodes".fuses.E6206CbVoltage24VOK )
      S_Coil( "Unit1.Alarms".systemFaultGeneral[26] )
   END_RUNG
   // the same network as SCL:
   IF NOT "Unit1.ControlNodes".fuses.E6206CbVoltage24VOK THEN
       "Unit1.Alarms".systemFaultGeneral[26] := TRUE;
   END_IF;
END_REGION

REGION Network 70: PFE System Fault General 27
   RUNG wire#powerrail
      I_Contact( "Unit1.ControlNodes".fuses.E6220CbVoltage24VOK )
      S_Coil( "Unit1.Alarms".systemFaultGeneral[27] )
   END_RUNG
   // the same network as SCL:
   IF NOT "Unit1.ControlNodes".fuses.E6220CbVoltage24VOK THEN
       "Unit1.Alarms".systemFaultGeneral[27] := TRUE;
   END_IF;
END_REGION

REGION Network 71: PFE System Fault General 28
   RUNG wire#powerrail
      I_Contact( "Unit1.ControlNodes".fuses.E6224CbVoltage24VOK )
      S_Coil( "Unit1.Alarms".systemFaultGeneral[28] )
   END_RUNG
   // the same network as SCL:
   IF NOT "Unit1.ControlNodes".fuses.E6224CbVoltage24VOK THEN
       "Unit1.Alarms".systemFaultGeneral[28] := TRUE;
   END_IF;
END_REGION

REGION Network 72: PFE System Fault General 29
   RUNG wire#powerrail
      I_Contact( "Unit1.ControlNodes".fuses.E6228CbVoltage24VOK )
      S_Coil( "Unit1.Alarms".systemFaultGeneral[29] )
   END_RUNG
   // the same network as SCL:
   IF NOT "Unit1.ControlNodes".fuses.E6228CbVoltage24VOK THEN
       "Unit1.Alarms".systemFaultGeneral[29] := TRUE;
   END_IF;
END_REGION

REGION Network 73: PFE System Fault General 30
   RUNG wire#powerrail
      I_Contact( "Unit1.ControlNodes".fuses.E6304CbVoltage24VOK )
      S_Coil( "Unit1.Alarms".systemFaultGeneral[30] )
   END_RUNG
   // the same network as SCL:
   IF NOT "Unit1.ControlNodes".fuses.E6304CbVoltage24VOK THEN
       "Unit1.Alarms".systemFaultGeneral[30] := TRUE;
   END_IF;
END_REGION

REGION Network 74: PFE System Fault General 31
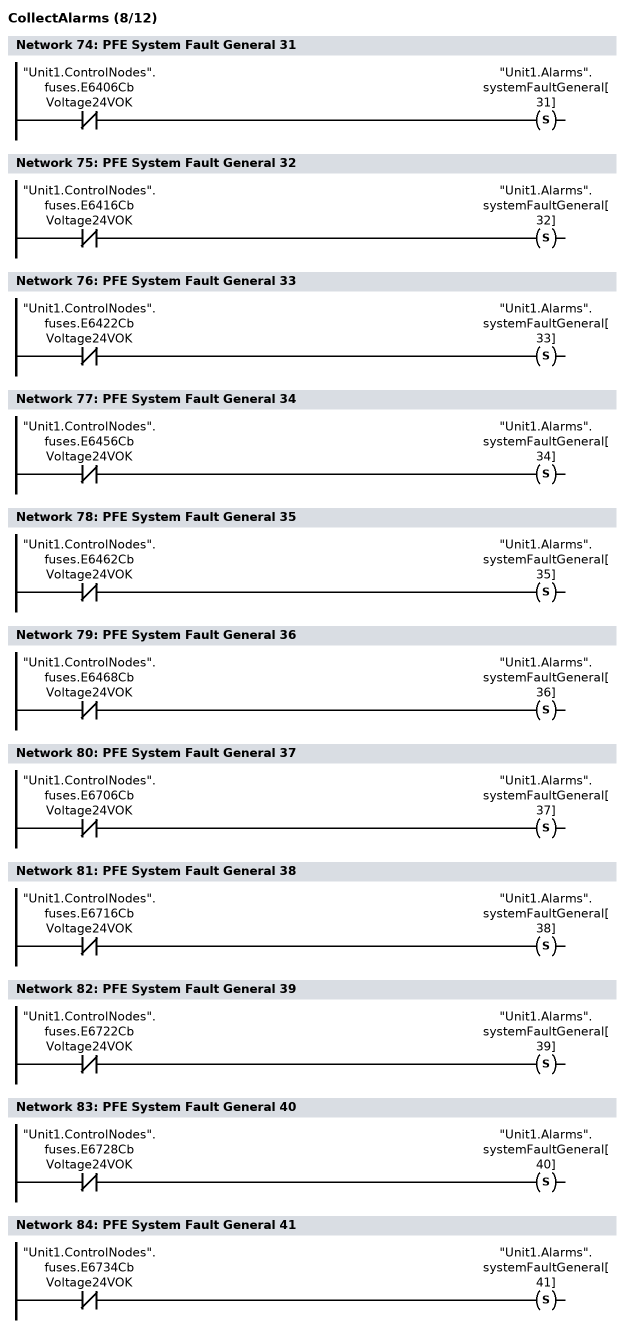
   RUNG wire#powerrail
      I_Contact( "Unit1.ControlNodes".fuses.E6406CbVoltage24VOK )
      S_Coil( "Unit1.Alarms".systemFaultGeneral[31] )
   END_RUNG
   // the same network as SCL:
   IF NOT "Unit1.ControlNodes".fuses.E6406CbVoltage24VOK THEN
       "Unit1.Alarms".systemFaultGeneral[31] := TRUE;
   END_IF;
END_REGION

REGION Network 75: PFE System Fault General 32
   RUNG wire#powerrail
      I_Contact( "Unit1.ControlNodes".fuses.E6416CbVoltage24VOK )
      S_Coil( "Unit1.Alarms".systemFaultGeneral[32] )
   END_RUNG
   // the same network as SCL:
   IF NOT "Unit1.ControlNodes".fuses.E6416CbVoltage24VOK THEN
       "Unit1.Alarms".systemFaultGeneral[32] := TRUE;
   END_IF;
END_REGION

REGION Network 76: PFE System Fault General 33
   RUNG wire#powerrail
      I_Contact( "Unit1.ControlNodes".fuses.E6422CbVoltage24VOK )
      S_Coil( "Unit1.Alarms".systemFaultGeneral[33] )
   END_RUNG
   // the same network as SCL:
   IF NOT "Unit1.ControlNodes".fuses.E6422CbVoltage24VOK THEN
       "Unit1.Alarms".systemFaultGeneral[33] := TRUE;
   END_IF;
END_REGION

REGION Network 77: PFE System Fault General 34
   RUNG wire#powerrail
      I_Contact( "Unit1.ControlNodes".fuses.E6456CbVoltage24VOK )
      S_Coil( "Unit1.Alarms".systemFaultGeneral[34] )
   END_RUNG
   // the same network as SCL:
   IF NOT "Unit1.ControlNodes".fuses.E6456CbVoltage24VOK THEN
       "Unit1.Alarms".systemFaultGeneral[34] := TRUE;
   END_IF;
END_REGION

REGION Network 78: PFE System Fault General 35
   RUNG wire#powerrail
      I_Contact( "Unit1.ControlNodes".fuses.E6462CbVoltage24VOK )
      S_Coil( "Unit1.Alarms".systemFaultGeneral[35] )
   END_RUNG
   // the same network as SCL:
   IF NOT "Unit1.ControlNodes".fuses.E6462CbVoltage24VOK THEN
       "Unit1.Alarms".systemFaultGeneral[35] := TRUE;
   END_IF;
END_REGION

REGION Network 79: PFE System Fault General 36
   RUNG wire#powerrail
      I_Contact( "Unit1.ControlNodes".fuses.E6468CbVoltage24VOK )
      S_Coil( "Unit1.Alarms".systemFaultGeneral[36] )
   END_RUNG
   // the same network as SCL:
   IF NOT "Unit1.ControlNodes".fuses.E6468CbVoltage24VOK THEN
       "Unit1.Alarms".systemFaultGeneral[36] := TRUE;
   END_IF;
END_REGION

REGION Network 80: PFE System Fault General 37
   RUNG wire#powerrail
      I_Contact( "Unit1.ControlNodes".fuses.E6706CbVoltage24VOK )
      S_Coil( "Unit1.Alarms".systemFaultGeneral[37] )
   END_RUNG
   // the same network as SCL:
   IF NOT "Unit1.ControlNodes".fuses.E6706CbVoltage24VOK THEN
       "Unit1.Alarms".systemFaultGeneral[37] := TRUE;
   END_IF;
END_REGION

REGION Network 81: PFE System Fault General 38
   RUNG wire#powerrail
      I_Contact( "Unit1.ControlNodes".fuses.E6716CbVoltage24VOK )
      S_Coil( "Unit1.Alarms".systemFaultGeneral[38] )
   END_RUNG
   // the same network as SCL:
   IF NOT "Unit1.ControlNodes".fuses.E6716CbVoltage24VOK THEN
       "Unit1.Alarms".systemFaultGeneral[38] := TRUE;
   END_IF;
END_REGION

REGION Network 82: PFE System Fault General 39
   RUNG wire#powerrail
      I_Contact( "Unit1.ControlNodes".fuses.E6722CbVoltage24VOK )
      S_Coil( "Unit1.Alarms".systemFaultGeneral[39] )
   END_RUNG
   // the same network as SCL:
   IF NOT "Unit1.ControlNodes".fuses.E6722CbVoltage24VOK THEN
       "Unit1.Alarms".systemFaultGeneral[39] := TRUE;
   END_IF;
END_REGION

REGION Network 83: PFE System Fault General 40
   RUNG wire#powerrail
      I_Contact( "Unit1.ControlNodes".fuses.E6728CbVoltage24VOK )
      S_Coil( "Unit1.Alarms".systemFaultGeneral[40] )
   END_RUNG
   // the same network as SCL:
   IF NOT "Unit1.ControlNodes".fuses.E6728CbVoltage24VOK THEN
       "Unit1.Alarms".systemFaultGeneral[40] := TRUE;
   END_IF;
END_REGION

REGION Network 84: PFE System Fault General 41
   RUNG wire#powerrail
      I_Contact( "Unit1.ControlNodes".fuses.E6734CbVoltage24VOK )
      S_Coil( "Unit1.Alarms".systemFaultGeneral[41] )
   END_RUNG
   // the same network as SCL:
   IF NOT "Unit1.ControlNodes".fuses.E6734CbVoltage24VOK THEN
       "Unit1.Alarms".systemFaultGeneral[41] := TRUE;
   END_IF;
END_REGION

REGION Network 85: PFE System Fault General 42
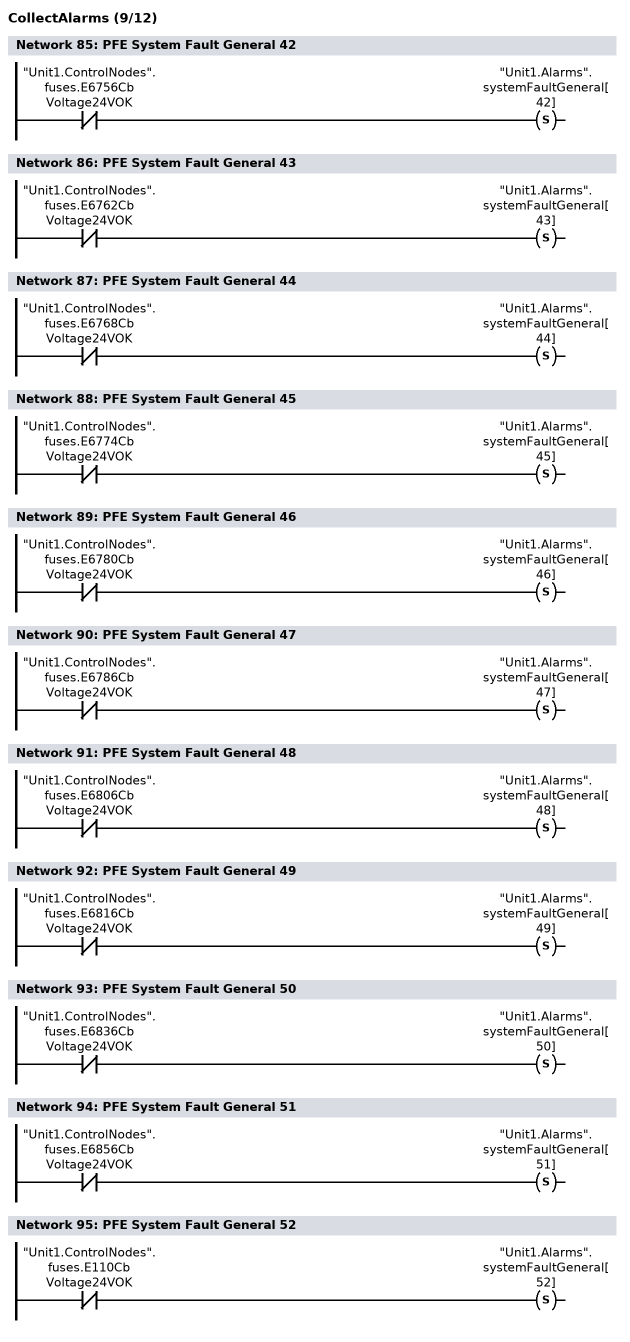
   RUNG wire#powerrail
      I_Contact( "Unit1.ControlNodes".fuses.E6756CbVoltage24VOK )
      S_Coil( "Unit1.Alarms".systemFaultGeneral[42] )
   END_RUNG
   // the same network as SCL:
   IF NOT "Unit1.ControlNodes".fuses.E6756CbVoltage24VOK THEN
       "Unit1.Alarms".systemFaultGeneral[42] := TRUE;
   END_IF;
END_REGION

REGION Network 86: PFE System Fault General 43
   RUNG wire#powerrail
      I_Contact( "Unit1.ControlNodes".fuses.E6762CbVoltage24VOK )
      S_Coil( "Unit1.Alarms".systemFaultGeneral[43] )
   END_RUNG
   // the same network as SCL:
   IF NOT "Unit1.ControlNodes".fuses.E6762CbVoltage24VOK THEN
       "Unit1.Alarms".systemFaultGeneral[43] := TRUE;
   END_IF;
END_REGION

REGION Network 87: PFE System Fault General 44
   RUNG wire#powerrail
      I_Contact( "Unit1.ControlNodes".fuses.E6768CbVoltage24VOK )
      S_Coil( "Unit1.Alarms".systemFaultGeneral[44] )
   END_RUNG
   // the same network as SCL:
   IF NOT "Unit1.ControlNodes".fuses.E6768CbVoltage24VOK THEN
       "Unit1.Alarms".systemFaultGeneral[44] := TRUE;
   END_IF;
END_REGION

REGION Network 88: PFE System Fault General 45
   RUNG wire#powerrail
      I_Contact( "Unit1.ControlNodes".fuses.E6774CbVoltage24VOK )
      S_Coil( "Unit1.Alarms".systemFaultGeneral[45] )
   END_RUNG
   // the same network as SCL:
   IF NOT "Unit1.ControlNodes".fuses.E6774CbVoltage24VOK THEN
       "Unit1.Alarms".systemFaultGeneral[45] := TRUE;
   END_IF;
END_REGION

REGION Network 89: PFE System Fault General 46
   RUNG wire#powerrail
      I_Contact( "Unit1.ControlNodes".fuses.E6780CbVoltage24VOK )
      S_Coil( "Unit1.Alarms".systemFaultGeneral[46] )
   END_RUNG
   // the same network as SCL:
   IF NOT "Unit1.ControlNodes".fuses.E6780CbVoltage24VOK THEN
       "Unit1.Alarms".systemFaultGeneral[46] := TRUE;
   END_IF;
END_REGION

REGION Network 90: PFE System Fault General 47
   RUNG wire#powerrail
      I_Contact( "Unit1.ControlNodes".fuses.E6786CbVoltage24VOK )
      S_Coil( "Unit1.Alarms".systemFaultGeneral[47] )
   END_RUNG
   // the same network as SCL:
   IF NOT "Unit1.ControlNodes".fuses.E6786CbVoltage24VOK THEN
       "Unit1.Alarms".systemFaultGeneral[47] := TRUE;
   END_IF;
END_REGION

REGION Network 91: PFE System Fault General 48
   RUNG wire#powerrail
      I_Contact( "Unit1.ControlNodes".fuses.E6806CbVoltage24VOK )
      S_Coil( "Unit1.Alarms".systemFaultGeneral[48] )
   END_RUNG
   // the same network as SCL:
   IF NOT "Unit1.ControlNodes".fuses.E6806CbVoltage24VOK THEN
       "Unit1.Alarms".systemFaultGeneral[48] := TRUE;
   END_IF;
END_REGION

REGION Network 92: PFE System Fault General 49
   RUNG wire#powerrail
      I_Contact( "Unit1.ControlNodes".fuses.E6816CbVoltage24VOK )
      S_Coil( "Unit1.Alarms".systemFaultGeneral[49] )
   END_RUNG
   // the same network as SCL:
   IF NOT "Unit1.ControlNodes".fuses.E6816CbVoltage24VOK THEN
       "Unit1.Alarms".systemFaultGeneral[49] := TRUE;
   END_IF;
END_REGION

REGION Network 93: PFE System Fault General 50
   RUNG wire#powerrail
      I_Contact( "Unit1.ControlNodes".fuses.E6836CbVoltage24VOK )
      S_Coil( "Unit1.Alarms".systemFaultGeneral[50] )
   END_RUNG
   // the same network as SCL:
   IF NOT "Unit1.ControlNodes".fuses.E6836CbVoltage24VOK THEN
       "Unit1.Alarms".systemFaultGeneral[50] := TRUE;
   END_IF;
END_REGION

REGION Network 94: PFE System Fault General 51
   RUNG wire#powerrail
      I_Contact( "Unit1.ControlNodes".fuses.E6856CbVoltage24VOK )
      S_Coil( "Unit1.Alarms".systemFaultGeneral[51] )
   END_RUNG
   // the same network as SCL:
   IF NOT "Unit1.ControlNodes".fuses.E6856CbVoltage24VOK THEN
       "Unit1.Alarms".systemFaultGeneral[51] := TRUE;
   END_IF;
END_REGION

REGION Network 95: PFE System Fault General 52
   RUNG wire#powerrail
      I_Contact( "Unit1.ControlNodes".fuses.E110CbVoltage24VOK )
      S_Coil( "Unit1.Alarms".systemFaultGeneral[52] )
   END_RUNG
   // the same network as SCL:
   IF NOT "Unit1.ControlNodes".fuses.E110CbVoltage24VOK THEN
       "Unit1.Alarms".systemFaultGeneral[52] := TRUE;
   END_IF;
END_REGION

REGION Network 96: PFE System Fault General 53
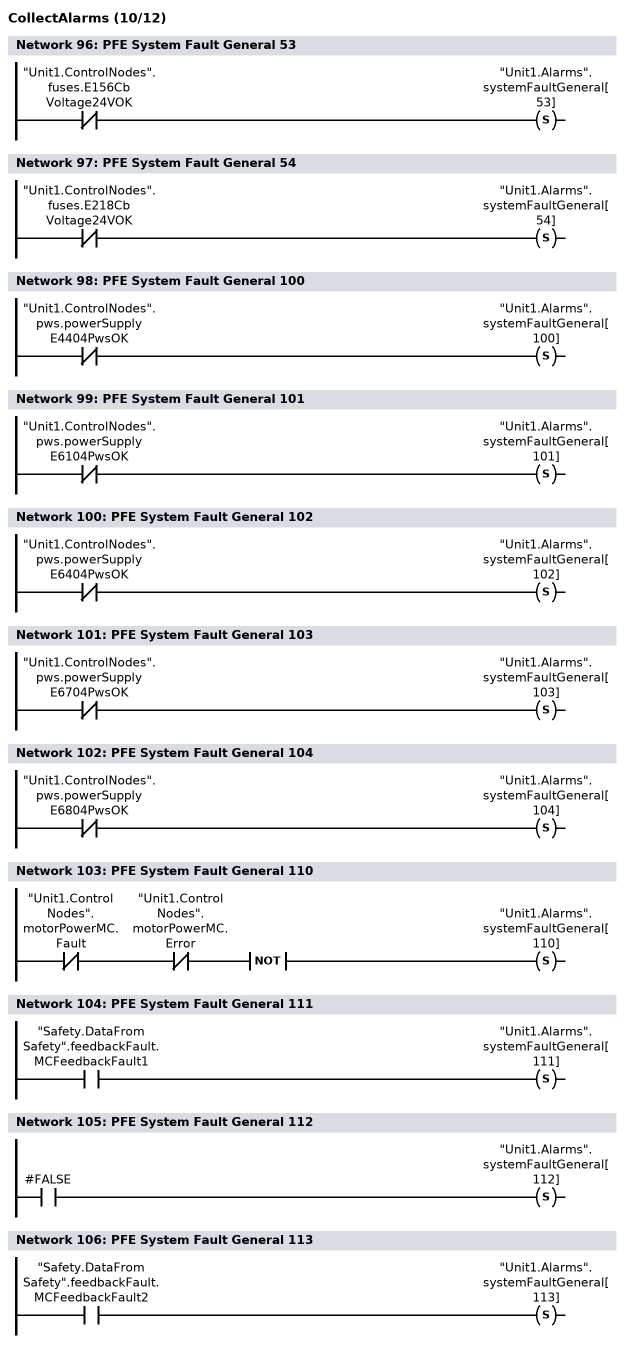
   RUNG wire#powerrail
      I_Contact( "Unit1.ControlNodes".fuses.E156CbVoltage24VOK )
      S_Coil( "Unit1.Alarms".systemFaultGeneral[53] )
   END_RUNG
   // the same network as SCL:
   IF NOT "Unit1.ControlNodes".fuses.E156CbVoltage24VOK THEN
       "Unit1.Alarms".systemFaultGeneral[53] := TRUE;
   END_IF;
END_REGION

REGION Network 97: PFE System Fault General 54
   RUNG wire#powerrail
      I_Contact( "Unit1.ControlNodes".fuses.E218CbVoltage24VOK )
      S_Coil( "Unit1.Alarms".systemFaultGeneral[54] )
   END_RUNG
   // the same network as SCL:
   IF NOT "Unit1.ControlNodes".fuses.E218CbVoltage24VOK THEN
       "Unit1.Alarms".systemFaultGeneral[54] := TRUE;
   END_IF;
END_REGION

REGION Network 98: PFE System Fault General 100
   RUNG wire#powerrail
      I_Contact( "Unit1.ControlNodes".pws.powerSupplyE4404PwsOK )
      S_Coil( "Unit1.Alarms".systemFaultGeneral[100] )
   END_RUNG
   // the same network as SCL:
   IF NOT "Unit1.ControlNodes".pws.powerSupplyE4404PwsOK THEN
       "Unit1.Alarms".systemFaultGeneral[100] := TRUE;
   END_IF;
END_REGION

REGION Network 99: PFE System Fault General 101
   RUNG wire#powerrail
      I_Contact( "Unit1.ControlNodes".pws.powerSupplyE6104PwsOK )
      S_Coil( "Unit1.Alarms".systemFaultGeneral[101] )
   END_RUNG
   // the same network as SCL:
   IF NOT "Unit1.ControlNodes".pws.powerSupplyE6104PwsOK THEN
       "Unit1.Alarms".systemFaultGeneral[101] := TRUE;
   END_IF;
END_REGION

REGION Network 100: PFE System Fault General 102
   RUNG wire#powerrail
      I_Contact( "Unit1.ControlNodes".pws.powerSupplyE6404PwsOK )
      S_Coil( "Unit1.Alarms".systemFaultGeneral[102] )
   END_RUNG
   // the same network as SCL:
   IF NOT "Unit1.ControlNodes".pws.powerSupplyE6404PwsOK THEN
       "Unit1.Alarms".systemFaultGeneral[102] := TRUE;
   END_IF;
END_REGION

REGION Network 101: PFE System Fault General 103
   RUNG wire#powerrail
      I_Contact( "Unit1.ControlNodes".pws.powerSupplyE6704PwsOK )
      S_Coil( "Unit1.Alarms".systemFaultGeneral[103] )
   END_RUNG
   // the same network as SCL:
   IF NOT "Unit1.ControlNodes".pws.powerSupplyE6704PwsOK THEN
       "Unit1.Alarms".systemFaultGeneral[103] := TRUE;
   END_IF;
END_REGION

REGION Network 102: PFE System Fault General 104
   RUNG wire#powerrail
      I_Contact( "Unit1.ControlNodes".pws.powerSupplyE6804PwsOK )
      S_Coil( "Unit1.Alarms".systemFaultGeneral[104] )
   END_RUNG
   // the same network as SCL:
   IF NOT "Unit1.ControlNodes".pws.powerSupplyE6804PwsOK THEN
       "Unit1.Alarms".systemFaultGeneral[104] := TRUE;
   END_IF;
END_REGION

REGION Network 103: PFE System Fault General 110
   RUNG wire#powerrail
      I_Contact( "Unit1.ControlNodes".motorPowerMC.Fault )
      I_Contact( "Unit1.ControlNodes".motorPowerMC.Error )
      Not()
      S_Coil( "Unit1.Alarms".systemFaultGeneral[110] )
   END_RUNG
   // the same network as SCL:
   IF NOT (NOT "Unit1.ControlNodes".motorPowerMC.Fault AND NOT "Unit1.ControlNodes".motorPowerMC.Error) THEN
       "Unit1.Alarms".systemFaultGeneral[110] := TRUE;
   END_IF;
END_REGION

REGION Network 104: PFE System Fault General 111
   RUNG wire#powerrail
      Contact( "Safety.DataFromSafety".feedbackFault.MCFeedbackFault1 )
      S_Coil( "Unit1.Alarms".systemFaultGeneral[111] )
   END_RUNG
   // the same network as SCL:
   IF "Safety.DataFromSafety".feedbackFault.MCFeedbackFault1 THEN
       "Unit1.Alarms".systemFaultGeneral[111] := TRUE;
   END_IF;
END_REGION

REGION Network 105: PFE System Fault General 112
   RUNG wire#powerrail
      Contact( #FALSE )
      S_Coil( "Unit1.Alarms".systemFaultGeneral[112] )
   END_RUNG
   // the same network as SCL:
   IF #FALSE THEN "Unit1.Alarms".systemFaultGeneral[112] := TRUE; END_IF;
END_REGION

REGION Network 106: PFE System Fault General 113
   RUNG wire#powerrail
      Contact( "Safety.DataFromSafety".feedbackFault.MCFeedbackFault2 )
      S_Coil( "Unit1.Alarms".systemFaultGeneral[113] )
   END_RUNG
   // the same network as SCL:
   IF "Safety.DataFromSafety".feedbackFault.MCFeedbackFault2 THEN
       "Unit1.Alarms".systemFaultGeneral[113] := TRUE;
   END_IF;
END_REGION

REGION Network 107: PFE System Fault General 114
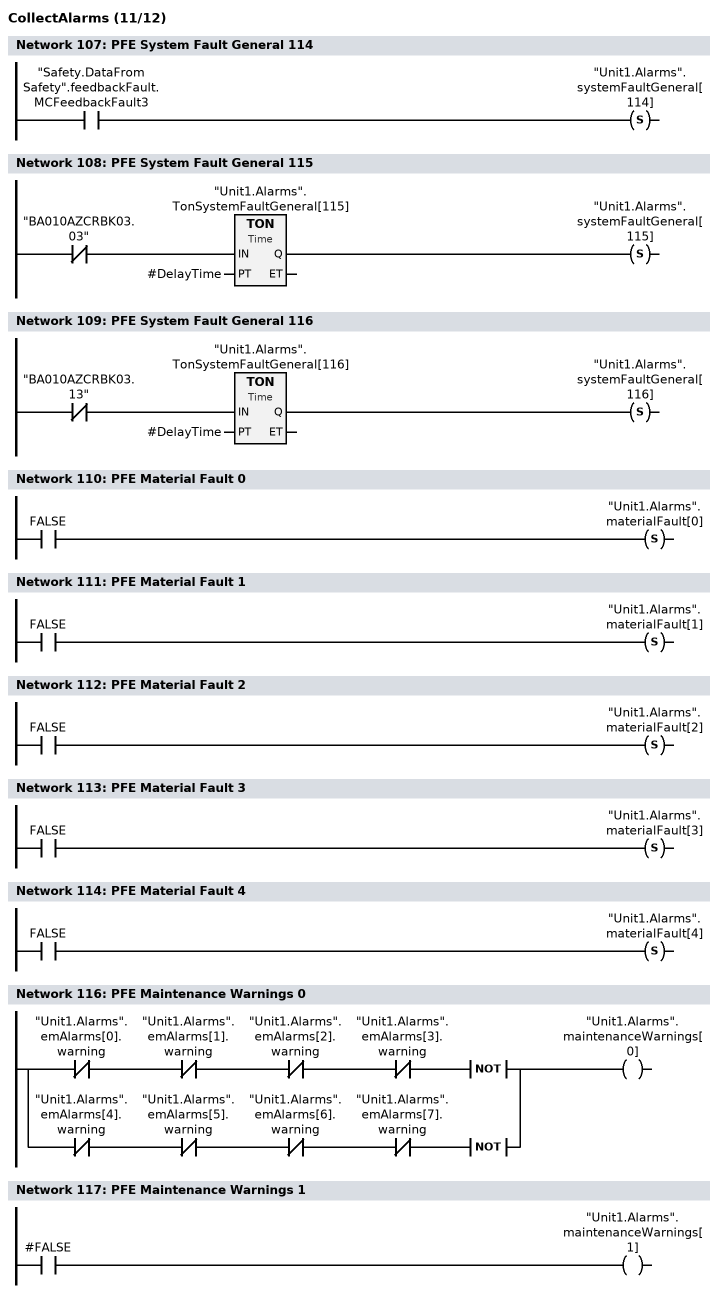
   RUNG wire#powerrail
      Contact( "Safety.DataFromSafety".feedbackFault.MCFeedbackFault3 )
      S_Coil( "Unit1.Alarms".systemFaultGeneral[114] )
   END_RUNG
   // the same network as SCL:
   IF "Safety.DataFromSafety".feedbackFault.MCFeedbackFault3 THEN
       "Unit1.Alarms".systemFaultGeneral[114] := TRUE;
   END_IF;
END_REGION

REGION Network 108: PFE System Fault General 115
   RUNG wire#powerrail
      I_Contact( "BA010AZCRBK03.03" )
      { S7_Templates := "time_type := Time" } "Unit1.Alarms".TonSystemFaultGeneral[115].TON(pt := #DelayTime, et =>)
      S_Coil( "Unit1.Alarms".systemFaultGeneral[115] )
   END_RUNG
   // the same network as SCL:
   "Unit1.Alarms".TonSystemFaultGeneral[115].TON(IN := NOT "BA010AZCRBK03.03", PT := #DelayTime);
   IF "Unit1.Alarms".TonSystemFaultGeneral[115].Q THEN
       "Unit1.Alarms".systemFaultGeneral[115] := TRUE;
   END_IF;
END_REGION

REGION Network 109: PFE System Fault General 116
   RUNG wire#powerrail
      I_Contact( "BA010AZCRBK03.13" )
      { S7_Templates := "time_type := Time" } "Unit1.Alarms".TonSystemFaultGeneral[116].TON(pt := #DelayTime, et =>)
      S_Coil( "Unit1.Alarms".systemFaultGeneral[116] )
   END_RUNG
   // the same network as SCL:
   "Unit1.Alarms".TonSystemFaultGeneral[116].TON(IN := NOT "BA010AZCRBK03.13", PT := #DelayTime);
   IF "Unit1.Alarms".TonSystemFaultGeneral[116].Q THEN
       "Unit1.Alarms".systemFaultGeneral[116] := TRUE;
   END_IF;
END_REGION

REGION Network 110: PFE Material Fault 0
   RUNG wire#powerrail
      Contact( FALSE )
      S_Coil( "Unit1.Alarms".materialFault[0] )
   END_RUNG
   // the same network as SCL:
   IF FALSE THEN "Unit1.Alarms".materialFault[0] := TRUE; END_IF;
END_REGION

REGION Network 111: PFE Material Fault 1
   RUNG wire#powerrail
      Contact( FALSE )
      S_Coil( "Unit1.Alarms".materialFault[1] )
   END_RUNG
   // the same network as SCL:
   IF FALSE THEN "Unit1.Alarms".materialFault[1] := TRUE; END_IF;
END_REGION

REGION Network 112: PFE Material Fault 2
   RUNG wire#powerrail
      Contact( FALSE )
      S_Coil( "Unit1.Alarms".materialFault[2] )
   END_RUNG
   // the same network as SCL:
   IF FALSE THEN "Unit1.Alarms".materialFault[2] := TRUE; END_IF;
END_REGION

REGION Network 113: PFE Material Fault 3
   RUNG wire#powerrail
      Contact( FALSE )
      S_Coil( "Unit1.Alarms".materialFault[3] )
   END_RUNG
   // the same network as SCL:
   IF FALSE THEN "Unit1.Alarms".materialFault[3] := TRUE; END_IF;
END_REGION

REGION Network 114: PFE Material Fault 4
   RUNG wire#powerrail
      Contact( FALSE )
      S_Coil( "Unit1.Alarms".materialFault[4] )
   END_RUNG
   // the same network as SCL:
   IF FALSE THEN "Unit1.Alarms".materialFault[4] := TRUE; END_IF;
END_REGION

REGION Network 115: *************** Warning **************************
END_REGION

REGION Network 116: PFE Maintenance Warnings 0
   RUNG wire#powerrail
      I_Contact( "Unit1.Alarms".emAlarms[0].warning )
      I_Contact( "Unit1.Alarms".emAlarms[1].warning )
      I_Contact( "Unit1.Alarms".emAlarms[2].warning )
      I_Contact( "Unit1.Alarms".emAlarms[3].warning )
      Not()
      wire#w1
      Coil( "Unit1.Alarms".maintenanceWarnings[0] )
   END_RUNG
   RUNG wire#powerrail
      I_Contact( "Unit1.Alarms".emAlarms[4].warning )
      I_Contact( "Unit1.Alarms".emAlarms[5].warning )
      I_Contact( "Unit1.Alarms".emAlarms[6].warning )
      I_Contact( "Unit1.Alarms".emAlarms[7].warning )
      Not()
   END_RUNG wire#w1
   // the same network as SCL:
   "Unit1.Alarms".maintenanceWarnings[0] := NOT (NOT "Unit1.Alarms".emAlarms[0].warning AND NOT "Unit1.Alarms".emAlarms[1].warning AND NOT "Unit1.Alarms".emAlarms[2].warning AND NOT "Unit1.Alarms".emAlarms[3].warning) OR NOT (NOT "Unit1.Alarms".emAlarms[4].warning AND NOT "Unit1.Alarms".emAlarms[5].warning AND NOT "Unit1.Alarms".emAlarms[6].warning AND NOT "Unit1.Alarms".emAlarms[7].warning);
END_REGION

REGION Network 117: PFE Maintenance Warnings 1
   RUNG wire#powerrail
      Contact( #FALSE )
      Coil( "Unit1.Alarms".maintenanceWarnings[1] )
   END_RUNG
   // the same network as SCL:
   "Unit1.Alarms".maintenanceWarnings[1] := #FALSE;
END_REGION

REGION Network 118: PFE Maintenance Warnings 10
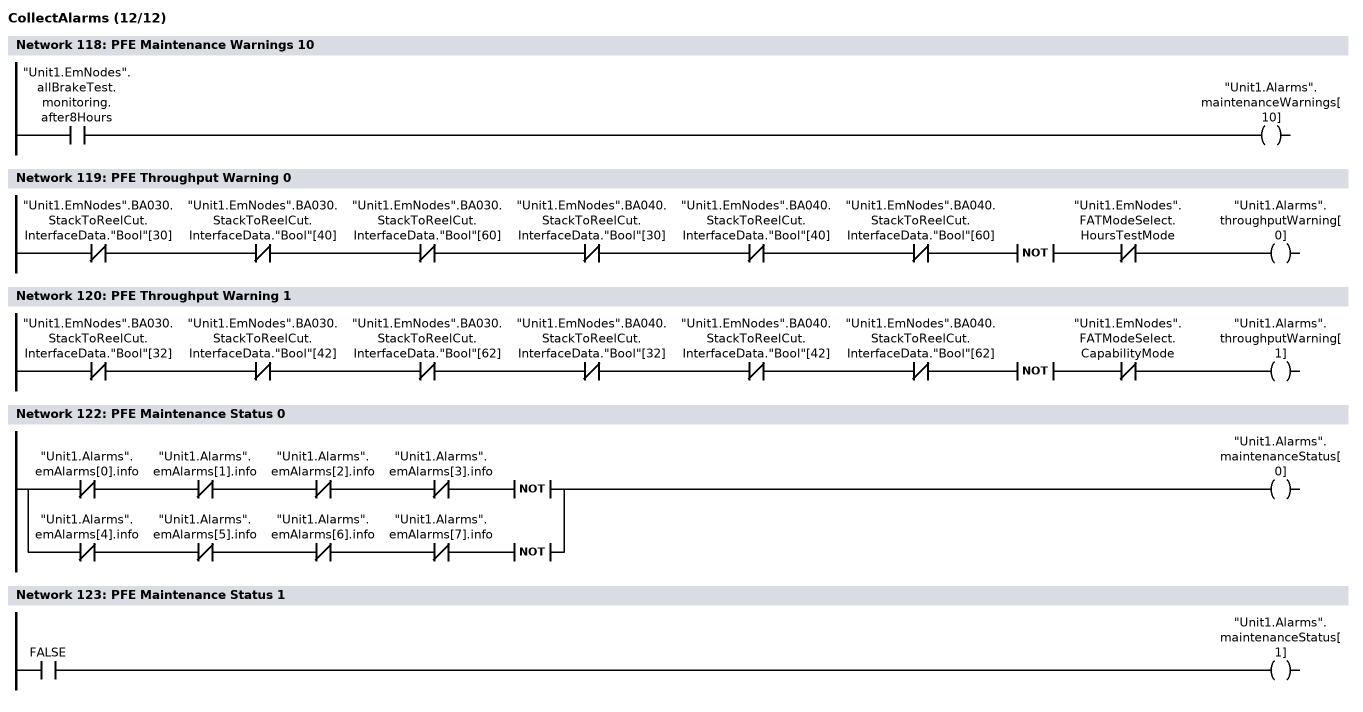
   RUNG wire#powerrail
      Contact( "Unit1.EmNodes".allBrakeTest.monitoring.after8Hours )
      Coil( "Unit1.Alarms".maintenanceWarnings[10] )
   END_RUNG
   // the same network as SCL:
   "Unit1.Alarms".maintenanceWarnings[10] := "Unit1.EmNodes".allBrakeTest.monitoring.after8Hours;
END_REGION

REGION Network 119: PFE Throughput Warning 0
   RUNG wire#powerrail
      I_Contact( "Unit1.EmNodes".BA030.StackToReelCut.InterfaceData."Bool"[30] )
      I_Contact( "Unit1.EmNodes".BA030.StackToReelCut.InterfaceData."Bool"[40] )
      I_Contact( "Unit1.EmNodes".BA030.StackToReelCut.InterfaceData."Bool"[60] )
      I_Contact( "Unit1.EmNodes".BA040.StackToReelCut.InterfaceData."Bool"[30] )
      I_Contact( "Unit1.EmNodes".BA040.StackToReelCut.InterfaceData."Bool"[40] )
      I_Contact( "Unit1.EmNodes".BA040.StackToReelCut.InterfaceData."Bool"[60] )
      Not()
      I_Contact( "Unit1.EmNodes".FATModeSelect.HoursTestMode )
      Coil( "Unit1.Alarms".throughputWarning[0] )
   END_RUNG
   // the same network as SCL:
   "Unit1.Alarms".throughputWarning[0] := NOT (NOT "Unit1.EmNodes".BA030.StackToReelCut.InterfaceData."Bool"[30] AND NOT "Unit1.EmNodes".BA030.StackToReelCut.InterfaceData."Bool"[40] AND NOT "Unit1.EmNodes".BA030.StackToReelCut.InterfaceData."Bool"[60] AND NOT "Unit1.EmNodes".BA040.StackToReelCut.InterfaceData."Bool"[30] AND NOT "Unit1.EmNodes".BA040.StackToReelCut.InterfaceData."Bool"[40] AND NOT "Unit1.EmNodes".BA040.StackToReelCut.InterfaceData."Bool"[60]) AND NOT "Unit1.EmNodes".FATModeSelect.HoursTestMode;
END_REGION

REGION Network 120: PFE Throughput Warning 1
   RUNG wire#powerrail
      I_Contact( "Unit1.EmNodes".BA030.StackToReelCut.InterfaceData."Bool"[32] )
      I_Contact( "Unit1.EmNodes".BA030.StackToReelCut.InterfaceData."Bool"[42] )
      I_Contact( "Unit1.EmNodes".BA030.StackToReelCut.InterfaceData."Bool"[62] )
      I_Contact( "Unit1.EmNodes".BA040.StackToReelCut.InterfaceData."Bool"[32] )
      I_Contact( "Unit1.EmNodes".BA040.StackToReelCut.InterfaceData."Bool"[42] )
      I_Contact( "Unit1.EmNodes".BA040.StackToReelCut.InterfaceData."Bool"[62] )
      Not()
      I_Contact( "Unit1.EmNodes".FATModeSelect.CapabilityMode )
      Coil( "Unit1.Alarms".throughputWarning[1] )
   END_RUNG
   // the same network as SCL:
   "Unit1.Alarms".throughputWarning[1] := NOT (NOT "Unit1.EmNodes".BA030.StackToReelCut.InterfaceData."Bool"[32] AND NOT "Unit1.EmNodes".BA030.StackToReelCut.InterfaceData."Bool"[42] AND NOT "Unit1.EmNodes".BA030.StackToReelCut.InterfaceData."Bool"[62] AND NOT "Unit1.EmNodes".BA040.StackToReelCut.InterfaceData."Bool"[32] AND NOT "Unit1.EmNodes".BA040.StackToReelCut.InterfaceData."Bool"[42] AND NOT "Unit1.EmNodes".BA040.StackToReelCut.InterfaceData."Bool"[62]) AND NOT "Unit1.EmNodes".FATModeSelect.CapabilityMode;
END_REGION

REGION Network 121: *************** Status ***************************
END_REGION

REGION Network 122: PFE Maintenance Status 0
   RUNG wire#powerrail
      I_Contact( "Unit1.Alarms".emAlarms[0].info )
      I_Contact( "Unit1.Alarms".emAlarms[1].info )
      I_Contact( "Unit1.Alarms".emAlarms[2].info )
      I_Contact( "Unit1.Alarms".emAlarms[3].info )
      Not()
      wire#w1
      Coil( "Unit1.Alarms".maintenanceStatus[0] )
   END_RUNG
   RUNG wire#powerrail
      I_Contact( "Unit1.Alarms".emAlarms[4].info )
      I_Contact( "Unit1.Alarms".emAlarms[5].info )
      I_Contact( "Unit1.Alarms".emAlarms[6].info )
      I_Contact( "Unit1.Alarms".emAlarms[7].info )
      Not()
   END_RUNG wire#w1
   // the same network as SCL:
   "Unit1.Alarms".maintenanceStatus[0] := NOT (NOT "Unit1.Alarms".emAlarms[0].info AND NOT "Unit1.Alarms".emAlarms[1].info AND NOT "Unit1.Alarms".emAlarms[2].info AND NOT "Unit1.Alarms".emAlarms[3].info) OR NOT (NOT "Unit1.Alarms".emAlarms[4].info AND NOT "Unit1.Alarms".emAlarms[5].info AND NOT "Unit1.Alarms".emAlarms[6].info AND NOT "Unit1.Alarms".emAlarms[7].info);
END_REGION

REGION Network 123: PFE Maintenance Status 1
   RUNG wire#powerrail
      Contact( FALSE )
      Coil( "Unit1.Alarms".maintenanceStatus[1] )
   END_RUNG
   // the same network as SCL:
   "Unit1.Alarms".maintenanceStatus[1] := FALSE;
END_REGION
END_FUNCTION
